FUNCTION_BLOCK "FB_FedExLoginResponse"
TITLE = FB_IDFWD
{ S7_Optimized_Access := 'TRUE' }
AUTHOR : MHSE
FAMILY : UPS_SpecificCommunication
VERSION : 3.0
// ATTRIBUTES
// AUTO_NUMBER = True
// BLOCK_NUMBER = 77
// END_ATTRIBUTES
//Function block to prepare and send the UPS IDFWD message.
   VAR_INPUT
      iUDT_Facility { ExternalAccessible := 'False'; ExternalVisible := 'False'; ExternalWritable := 'False'} : "UDT_FedExFacility";   // System configuration
      is_LastHost { ExternalAccessible := 'False'; ExternalVisible := 'False'; ExternalWritable := 'False'} : String;   // IP Address of the existing connection. If this isthe first connection, IP Address or Hostname
      ix_ConnectionStatus { ExternalAccessible := 'False'; ExternalVisible := 'False'; ExternalWritable := 'False'} : Bool;   // 1- Success, 0- Failure
   END_VAR

   VAR_OUTPUT
      qx_Error { ExternalAccessible := 'False'; ExternalVisible := 'False'; ExternalWritable := 'False'} : Bool;   // Collective error output
   END_VAR

   VAR_IN_OUT
      iqUDT_FifoHeader : "UDT_FifoHeader";   // FIFO header
      iqa_FifoData : Array[*] of "UDT_Message";   // FIFO data
   END_VAR

   VAR
      s_R_TRIG_LoginRequest {InstructionName := 'R_TRIG'; LibVersion := '1.0'; ExternalAccessible := 'False'; ExternalVisible := 'False'; ExternalWritable := 'False'; S7_SetPoint := 'False'} : R_TRIG;   // R_TRIG send login responde messge
      s_UDT_MessageArray { ExternalAccessible := 'False'; ExternalVisible := 'False'; ExternalWritable := 'False'; S7_SetPoint := 'False'} : "UDT_Message";   // Message character array
      sa_Status { ExternalAccessible := 'False'; ExternalVisible := 'False'; ExternalWritable := 'False'} : Struct   // Status structure
         FIFOStatus { ExternalAccessible := 'False'; ExternalVisible := 'False'; ExternalWritable := 'False'} : "UDT_FifoStatus";   //  FIFO Status structure
         FIFOError { ExternalAccessible := 'False'; ExternalVisible := 'False'; ExternalWritable := 'False'; S7_SetPoint := 'True'} : Bool;   //  FIFO error
         FIFOWarning { ExternalAccessible := 'False'; ExternalVisible := 'False'; ExternalWritable := 'False'; S7_SetPoint := 'True'} : Bool;   //  FIFO warning
         InvalidSystemIDLen { ExternalAccessible := 'False'; ExternalVisible := 'False'; ExternalWritable := 'False'} : Bool;   //  Invalid designated system parameter input
         InvalidFacialityIDLen { ExternalAccessible := 'False'; ExternalVisible := 'False'; ExternalWritable := 'False'} : Bool;   //  Invalid GIN
         InvalidMsgArraySize { ExternalAccessible := 'False'; ExternalVisible := 'False'; ExternalWritable := 'False'} : Bool;   //  Invalid message array size
      END_STRUCT;
      ss_Message { ExternalAccessible := 'False'; ExternalVisible := 'False'; ExternalWritable := 'False'} : String;   // Message character string
      ss_ConnectionStatus { ExternalAccessible := 'False'; ExternalVisible := 'False'; ExternalWritable := 'False'} : String;   // Connection status. Y- Sucess, N- Failure
      ss_LastHost { ExternalAccessible := 'False'; ExternalVisible := 'False'; ExternalWritable := 'False'} : String;   // Last host IP adress
      ss_VersionID { ExternalAccessible := 'False'; ExternalVisible := 'False'; ExternalWritable := 'False'} : String;   // Version ID
      sui_MsgArrayElNr { ExternalAccessible := 'False'; ExternalVisible := 'False'; ExternalWritable := 'False'} : UInt;   // Number of written message characters
      si_MaxMsgLen { ExternalAccessible := 'False'; ExternalVisible := 'False'; ExternalWritable := 'False'} : Int;   // Maximum message length
      si_MsgLen { ExternalAccessible := 'False'; ExternalVisible := 'False'; ExternalWritable := 'False'} : Int;   // String character message length
      si_FacialityIDLen { ExternalAccessible := 'False'; ExternalVisible := 'False'; ExternalWritable := 'False'} : Int;   // Faciality ID length
      si_SystemIDLen { ExternalAccessible := 'False'; ExternalVisible := 'False'; ExternalWritable := 'False'} : Int;   // System ID length
      si_VersionIDLen { ExternalAccessible := 'False'; ExternalVisible := 'False'; ExternalWritable := 'False'} : Int;   // Version ID length
      si_i { ExternalAccessible := 'False'; ExternalVisible := 'False'; ExternalWritable := 'False'} : Int;   // Loop counter
      si_LastHostLen { ExternalAccessible := 'False'; ExternalVisible := 'False'; ExternalWritable := 'False'} : Int;   // Last host field length
      si_j { ExternalAccessible := 'False'; ExternalVisible := 'False'; ExternalWritable := 'False'} : Int;   // Loop counter
   END_VAR

   VAR CONSTANT
      cc_NULL : Char := '$00';   // NULL sign
      cc_STX : Char := '$02';   // Message type
      cc_ETX : Char := '$03';   // End of the text
      cs_MessageLength : String := '0066';   // Start of the text
      cs_MessageType : String := 'LR';   // Legth of the message
   END_VAR


BEGIN
	(*
	----------------------------------------------------------------------------------------

	Version history:
	Date        | Version   | Author        | Remark
	----------------------------------------------------------------------------------------
	30/06/2021  | 1.0       | J.Krawczuk    | first release MHS TIA 16.0
	16/11/2021  | 1.2       | M.Piela       | Updating regions numbering and interface changes
	21/02/2023  | 4.0       | F.Baten       | 4.0 Release TIA 17.5
	*)

	REGION 1 – FIFO header status update

	    // Mode 'S' - FIFO register status update
	    "FC_Fifo"(ic_Mode := 'S',
	              qUDT_Status => #sa_Status.FIFOStatus,
	              qx_Error => #sa_Status.FIFOError,
	              qx_Warning => #sa_Status.FIFOWarning,
	              iqv_Data := #s_UDT_MessageArray,
	              iqUDT_FifoHeader := #iqUDT_FifoHeader,
	              iqv_DataBuffer := #iqa_FifoData);

	END_REGION

	REGION 2 – Configuration check and create error

	    #si_FacialityIDLen := LEN(#iUDT_Facility.FacilityID);
	    #si_SystemIDLen := LEN(#iUDT_Facility.SystemID);

	    #sa_Status.InvalidSystemIDLen := #si_SystemIDLen <> 15;
	    #sa_Status.InvalidFacialityIDLen := #si_FacialityIDLen <> 6;

	END_REGION

	REGION 3 – Message preparation


	    IF (NOT #iqUDT_FifoHeader.Status.Full)                         // FIFO isn't full
	    THEN
	        IF (NOT #sa_Status.FIFOError                                // No FIFO errors
	            AND NOT #sa_Status.InvalidSystemIDLen                   // Length of system ID field is ok
	            AND NOT #sa_Status.InvalidFacialityIDLen)               // Length of faciality ID field is ok

	        THEN
	            REGION 3.1 – Message preparation

	                IF #ix_ConnectionStatus                             //Creating connection status
	                THEN
	                    #ss_ConnectionStatus := 'Y';

	                ELSE
	                    #ss_ConnectionStatus := 'N';

	                END_IF;

	                #ss_LastHost := '';                                 // Initializing Last host field
	                #ss_LastHost := #is_LastHost;
	                #si_LastHostLen := LEN(#ss_LastHost);

	                // Filling up rest of the field with spaces
	                FOR #si_i := 1 TO 32 - #si_LastHostLen DO

	                    #ss_LastHost := CONCAT(IN1 := #ss_LastHost,
	                                           IN2 := ' ');

	                END_FOR;

	                #ss_VersionID := '';                                // Initializing Version ID field
	                #ss_VersionID := #iUDT_Facility.VersionID;
	                #si_VersionIDLen := LEN(#ss_VersionID);

	                // Filling up rest of the field with space
	                FOR #si_j := 1 TO 6 - #si_VersionIDLen DO

	                    #ss_VersionID := CONCAT(IN1 := #ss_VersionID,
	                                            IN2 := ' ');

	                END_FOR;

	                // Message preparation

	                // Login Response message composing according to the structure
	                #ss_Message := CONCAT(IN1 := #cc_STX,                               // Start of the message (STX) '$02'
	                                      IN2 := #cs_MessageLength,                     // Message length
	                                      IN3 := #cs_MessageType,                       // Message type
	                                      IN4 := #iUDT_Facility.FacilityID,           // Facility ID
	                                      IN5 := #iUDT_Facility.SystemID,             // System ID
	                                      IN6 := #ss_VersionID,                         // Used version ID
	                                      IN7 := #ss_ConnectionStatus,                  // Connection status
	                                      IN8 := #ss_LastHost,                          // Last connected host IP adress
	                                      IN9 := #cc_ETX);                              // End of the message (ETX) '$03"

	            END_REGION

	            REGION 3.2 – Maximum number of the message characters

	                #si_MaxMsgLen := "FC_GetNrOfArrayEl"(iv_Array := #s_UDT_MessageArray.Character);

	            END_REGION

	            REGION 3.3 – Length of the complete message

	                #si_MsgLen := LEN(#ss_Message);

	            END_REGION

	            REGION 3.4 –  Message array size validation

	                #sa_Status.InvalidMsgArraySize := #si_MsgLen > #si_MaxMsgLen;

	            END_REGION

	            REGION 3.5 –  Message character string conversion to a message array of characters

	                IF (NOT #sa_Status.InvalidMsgArraySize)                 // Message character array size is valid
	                THEN

	                    Strg_TO_Chars(Strg := #ss_Message,
	                                  pChars := 0,
	                                  Cnt => #sui_MsgArrayElNr,
	                                  Chars := #s_UDT_MessageArray.Character);

	                END_IF;

	            END_REGION

	            REGION 3.6 – Clearing remaining characters in the message character array

	                IF (NOT #sa_Status.InvalidMsgArraySize)                 // Message character array size is valid
	                THEN

	                    // Filling up not used message character array elements with ' '
	                    FILL_BLK(IN := #cc_NULL,
	                             COUNT := UINT_TO_ULINT(INT_TO_UINT(#si_MaxMsgLen) - #sui_MsgArrayElNr),
	                             OUT => #s_UDT_MessageArray.Character[#sui_MsgArrayElNr]);

	                END_IF;

	            END_REGION


	            REGION 3.7 – Message write into a FIFO register

	                IF (NOT #sa_Status.InvalidMsgArraySize)      // Message character array size is valid
	                THEN

	                    // Mode 'W' - Write FIFO record
	                    "FC_Fifo"(ic_Mode := 'W',
	                              qUDT_Status => #sa_Status.FIFOStatus,
	                              qx_Error => #sa_Status.FIFOError,
	                              qx_Warning => #sa_Status.FIFOWarning,
	                              iqv_Data := #s_UDT_MessageArray,
	                              iqUDT_FifoHeader := #iqUDT_FifoHeader,
	                              iqv_DataBuffer := #iqa_FifoData);

	                END_IF;

	            END_REGION

	        END_IF;

	        // In case of FIFO full, the FIFO full error bit and FIFO collective error bit are set
	    ELSE
	        #sa_Status.FIFOError := TRUE;
	        #sa_Status.FIFOStatus.FifoFull := TRUE;

	    END_IF;

	END_REGION

	REGION 4 – Status

	    // Parametrization collective error output
	    #qx_Error :=
	    #sa_Status.InvalidSystemIDLen                               // Invalid System ID string length
	    OR #sa_Status.InvalidFacialityIDLen                         // Invalid Faciality ID lenght
	    OR #sa_Status.InvalidMsgArraySize                           // Invalid message array size
	    OR #sa_Status.FIFOError;                                    // FIFO error

	END_REGION
END_FUNCTION_BLOCK

FUNCTION_BLOCK "FB_FedExEquipmentStatusMessage"
TITLE = FB_Heartbeat
{ S7_Optimized_Access := 'TRUE' }
AUTHOR : MHSE
FAMILY : UPS_SpecificCommunication
VERSION : 3.0
// ATTRIBUTES
// AUTO_NUMBER = True
// BLOCK_NUMBER = 72
// END_ATTRIBUTES
//Function block to send and monitor the UPS heartbeat message.
   VAR_INPUT
      iUDT_Facility { ExternalAccessible := 'False'; ExternalVisible := 'False'; ExternalWritable := 'False'} : "UDT_FedExFacility";   // System configuration
      is_LOConEquipment { ExternalAccessible := 'False'; ExternalVisible := 'False'; ExternalWritable := 'False'} : String[3];   // Location of the equipment
      is_DEPCOD { ExternalAccessible := 'False'; ExternalVisible := 'False'; ExternalWritable := 'False'} : String[6];   // Depot Code
      is_TYPofEquipment { ExternalAccessible := 'False'; ExternalVisible := 'False'; ExternalWritable := 'False'} : String[3];   // Type of equipment
      is_NumberOfTheEquipment { ExternalAccessible := 'False'; ExternalVisible := 'False'; ExternalWritable := 'False'} : String[3];   // Number of the equipment 001-999
      is_DeviceType { ExternalAccessible := 'False'; ExternalVisible := 'False'; ExternalWritable := 'False'} : String[6];   // Type of Device
      is_DeviceID { ExternalAccessible := 'False'; ExternalVisible := 'False'; ExternalWritable := 'False'} : String[6];   // ID of the Device Type
      is_StatusCode { ExternalAccessible := 'False'; ExternalVisible := 'False'; ExternalWritable := 'False'} : String[3];   // Status code values
   END_VAR

   VAR_OUTPUT
      qx_Error { ExternalAccessible := 'False'; ExternalVisible := 'False'; ExternalWritable := 'False'} : Bool;   // Error
   END_VAR

   VAR_IN_OUT
      iqUDT_FifoHeader : "UDT_FifoHeader";   // FIFO header
      iqa_FifoData : Array[*] of "UDT_Message";   // FIFO data
   END_VAR

   VAR
      sUDT_MessageArray { ExternalAccessible := 'False'; ExternalVisible := 'False'; ExternalWritable := 'False'; S7_SetPoint := 'False'} : "UDT_Message";   // Message character array
      sa_Status { ExternalAccessible := 'False'; ExternalVisible := 'False'; ExternalWritable := 'False'} : Struct   // Status structure
         FIFOStatus { ExternalAccessible := 'False'; ExternalVisible := 'False'; ExternalWritable := 'False'} : "UDT_FifoStatus";   // FIFO status structure
         FIFOError { ExternalAccessible := 'False'; ExternalVisible := 'False'; ExternalWritable := 'False'; S7_SetPoint := 'True'} : Bool;   // FIFO data buffer full
         FIFOWarning { ExternalAccessible := 'False'; ExternalVisible := 'False'; ExternalWritable := 'False'; S7_SetPoint := 'True'} : Bool;   // FIFO error
         InvalidGIN { ExternalAccessible := 'False'; ExternalVisible := 'False'; ExternalWritable := 'False'} : Bool;   //  Invalid GIN
         InvalidMessageLength { ExternalAccessible := 'False'; ExternalVisible := 'False'; ExternalWritable := 'False'} : Bool;   //  Invalid PLC ID or TRAY ID
         InvalidMsgArraySize { ExternalAccessible := 'False'; ExternalVisible := 'False'; ExternalWritable := 'False'} : Bool;   // Heartbeat timeout lower than zero or lower than heartbeat time interval
      END_STRUCT;
      ss_LLCSystemID { ExternalAccessible := 'False'; ExternalVisible := 'False'; ExternalWritable := 'False'} : String[15];   // Identifier of Low-Level controls
      ss_DeviceID { ExternalAccessible := 'False'; ExternalVisible := 'False'; ExternalWritable := 'False'} : String[6];
      ss_DeviceType { ExternalAccessible := 'False'; ExternalVisible := 'False'; ExternalWritable := 'False'} : String[6];
      ss_StatusCode { ExternalAccessible := 'False'; ExternalVisible := 'False'; ExternalWritable := 'False'} : String[3];
      ss_Message { ExternalAccessible := 'False'; ExternalVisible := 'False'; ExternalWritable := 'False'} : String;   // Message character string
      sui_MsgArrayElNr { ExternalAccessible := 'False'; ExternalVisible := 'False'; ExternalWritable := 'False'} : UInt;   // Invalid message array size
      si_MaxMsgLen { ExternalAccessible := 'False'; ExternalVisible := 'False'; ExternalWritable := 'False'} : Int;   // Maximum message length
      si_MsgLen { ExternalAccessible := 'False'; ExternalVisible := 'False'; ExternalWritable := 'False'} : Int;   // String character message length
      si_LostMsg { ExternalAccessible := 'False'; ExternalVisible := 'False'; ExternalWritable := 'False'} : Int;   // Number of lost messages
      si_DeviceIDLen { ExternalAccessible := 'False'; ExternalVisible := 'False'; ExternalWritable := 'False'} : Int;
      si_DeviceTypeLen { ExternalAccessible := 'False'; ExternalVisible := 'False'; ExternalWritable := 'False'} : Int;
      si_StatusCodeLen { ExternalAccessible := 'False'; ExternalVisible := 'False'; ExternalWritable := 'False'} : Int;
      si_LenFillLoop { ExternalAccessible := 'False'; ExternalVisible := 'False'; ExternalWritable := 'False'} : Int;   // Loop couter
      sx_MsgLost { ExternalAccessible := 'False'; ExternalVisible := 'False'; ExternalWritable := 'False'} : Bool;   // Message lost
   END_VAR

   VAR CONSTANT
      cc_NULL : Char := '$00';   // NULL sign
      cc_STX : Char := '$02';   // Start of the text
      cc_ETX : Char := '$03';   // End of the text
      cs_Length : String := '0058';   // Legth of the message
      cs_MessageType : String := 'ES';   // Message type
   END_VAR


BEGIN
	(*
	----------------------------------------------------------------------------------------

	Version history:
	Date        | Version   | Author        | Remark
	----------------------------------------------------------------------------------------
	24/05/2019  | 0.1       | L.Klar        | first release MHS TIA 15.1
	29/06/2021  | 1.0       | F.Baten       | first release MHS TIA 16.4
	10/11/2021  | 1.2       | M.Piela       | Updating regions numbering, interface changes
	10/11/2021  | 1.3       | M.Piela       | Device ID, Device Type and Status Code conversion
	21/02/2023  | 4.0       | F.Baten       | 4.0 Release TIA 17.5
	*)

	REGION 1 – FIFO header status update

	    // Mode 'S' - FIFO register status update
	    "FC_Fifo"(ic_Mode := 'S',
	              qUDT_Status => #sa_Status.FIFOStatus,
	              qx_Error => #sa_Status.FIFOError,
	              qx_Warning => #sa_Status.FIFOWarning,
	              iqv_Data := #sUDT_MessageArray,
	              iqUDT_FifoHeader := #iqUDT_FifoHeader,
	              iqv_DataBuffer := #iqa_FifoData);
	END_REGION

	REGION 2 – Message preparation

	    IF NOT #iqUDT_FifoHeader.Status.Full                 // FIFO isn't full
	    THEN

	        REGION 2.1 - LLC System ID
	            #ss_LLCSystemID := CONCAT(IN1 := #is_DEPCOD,
	                                      IN2 := #is_LOConEquipment,
	                                      IN3 := #is_TYPofEquipment,
	                                      IN4 := #is_NumberOfTheEquipment);
	        END_REGION

	        REGION 2.2. Device Type

	            #ss_DeviceType := #is_DeviceType;
	            #si_DeviceTypeLen := LEN(#ss_DeviceType);

	            IF #si_DeviceTypeLen < 6
	            THEN
	                FOR #si_LenFillLoop := #si_DeviceTypeLen TO 6 DO
	                    #ss_DeviceType := CONCAT(IN1 := #ss_DeviceType,
	                                             IN2 := ' ');
	                END_FOR;

	            END_IF;

	        END_REGION

	        REGION 2.3. Device ID

	            #ss_DeviceID := #is_DeviceID;
	            #si_DeviceIDLen := LEN(#ss_DeviceID);

	            IF #si_DeviceIDLen < 6
	            THEN
	                FOR #si_LenFillLoop := #si_DeviceIDLen TO 6 DO
	                    #ss_DeviceID := CONCAT(IN1 := #ss_DeviceID,
	                                           IN2 := ' ');
	                END_FOR;

	            END_IF;

	        END_REGION

	        REGION 2.4. Status Code

	            #ss_StatusCode := #is_StatusCode;
	            #si_StatusCodeLen := LEN(#ss_StatusCode);

	            IF #si_StatusCodeLen < 3
	            THEN
	                FOR #si_LenFillLoop := #si_StatusCodeLen TO 3 DO
	                    #ss_StatusCode := CONCAT(IN1 := #ss_StatusCode,
	                                             IN2 := ' ');
	                END_FOR;

	            END_IF;

	        END_REGION

	        IF NOT #sa_Status.FIFOError                   // No FIFO error
	        THEN
	            REGION 2.5 – Message preparation
	                // Message composing according to the structure: STX,Body ,ETX
	                #ss_Message := CONCAT(IN1 := #cc_STX,
	                                      IN2 := #cs_Length,
	                                      IN3 := #cs_MessageType,
	                                      IN4 := #ss_LLCSystemID,
	                                      IN5 := #ss_DeviceType,
	                                      IN6 := #ss_DeviceID,
	                                      IN7 := #ss_StatusCode,
	                                      IN8 := "DB_Time".Timestamp,
	                                      IN9 := #iUDT_Facility.TimeZoneDesignator,
	                                      IN10 := #cc_ETX);

	            END_REGION

	            REGION 2.6 – Maximum number of the message characters

	                #si_MaxMsgLen := "FC_GetNrOfArrayEl"(iv_Array := #sUDT_MessageArray.Character);

	            END_REGION

	            REGION 2.7 – Length of the complete message

	                #si_MsgLen := LEN(#ss_Message);
	                // Message length validation
	                #sa_Status.InvalidMessageLength := #si_MsgLen - 2 <> STRING_TO_INT(#cs_Length);

	            END_REGION

	            REGION 2.8 –  Message array size validation

	                #sa_Status.InvalidMsgArraySize := #si_MsgLen > #si_MaxMsgLen;

	            END_REGION

	            REGION 2.9 –  Message character string conversion to a message array of characters

	                IF (NOT #sa_Status.InvalidMsgArraySize)     // Message character array size is valid
	                THEN

	                    Strg_TO_Chars(Strg := #ss_Message,
	                                  pChars := 0,
	                                  Cnt => #sui_MsgArrayElNr,
	                                  Chars := #sUDT_MessageArray.Character);

	                END_IF;

	            END_REGION

	            REGION 2.10 – Clearing remaining characters in the message character array

	                IF (NOT #sa_Status.InvalidMsgArraySize)     // Message character array size is valid
	                THEN

	                    // Filling up not used message character array elements with '$00' (ASCII - 16#00)
	                    FILL_BLK(IN := #cc_NULL,
	                             COUNT := UINT_TO_ULINT(INT_TO_UINT(#si_MaxMsgLen) - #sui_MsgArrayElNr),
	                             OUT => #sUDT_MessageArray.Character[#sui_MsgArrayElNr]);

	                END_IF;

	            END_REGION

	            REGION 2.11 – Message write into a FIFO register

	                IF NOT #sa_Status.InvalidMsgArraySize      // Message character array size is valid
	                THEN

	                    // Mode 'W' - Write FIFO record
	                    "FC_Fifo"(ic_Mode := 'W',
	                              qUDT_Status => #sa_Status.FIFOStatus,
	                              qx_Error => #sa_Status.FIFOError,
	                              qx_Warning => #sa_Status.FIFOWarning,
	                              iqv_Data := #sUDT_MessageArray,
	                              iqUDT_FifoHeader := #iqUDT_FifoHeader,
	                              iqv_DataBuffer := #iqa_FifoData);
	                END_IF;

	            END_REGION

	        END_IF;

	        // In case of FIFO full, the FIFO full error bit and FIFO collective error bit are set
	    ELSE

	        #sa_Status.FIFOError := TRUE;
	        #sa_Status.FIFOStatus.FifoFull := TRUE;

	    END_IF;

	END_REGION

	REGION 3 - Writing output

	    #qx_Error := #sa_Status.InvalidMessageLength        // Invalid message length
	    OR #sa_Status.InvalidMsgArraySize                   // Invalid message array size
	    OR #sa_Status.FIFOError;                            // FIFO error

	END_REGION
END_FUNCTION_BLOCK

FUNCTION "FC_Statistics" : Void
TITLE = FC_Statistics
{ S7_Optimized_Access := 'TRUE' }
AUTHOR : MHSE
FAMILY : GeneralSystemFunctions
VERSION : 3.0
// ATTRIBUTES
// AUTO_NUMBER = True
// BLOCK_NUMBER = 26
// END_ATTRIBUTES
//Function to calculate statistics.
   VAR_INPUT
      ix_Reset : Bool;   // Reset statistics data
      ix_Activate : Bool;   // Activete statistics counters
      ix_RTrigActivate : Bool;   // Activation rise trigger
   END_VAR

   VAR_IN_OUT
      iqUDT_Statistics : "UDT_EventStatistic";   // Statistic structure
   END_VAR


BEGIN
	(*
	----------------------------------------------------------------------------------------

	Version history:
	Date        | Version   | Author        | Remark
	----------------------------------------------------------------------------------------
	24/05/2019  | 0.1       | C. Leite      | first release MHS TIA 15.1
	17/07/2019  | 0.2       | A.Nowak       | Add comments
	24/07/2019  | 2.0       | L.Klar        | 2.0 MHS library release TIA 15.1
	27/08/2019  | 2.1       | M.Kurpiers    | Comments adjusted
	04/11/2019  | 2.2       | L.Klar        | 1 second pulse changed from memory bit to DB variable
	12/11/2019  | 3.0       | P.Majka       | 3.0 MHS library release TIA 15.1
	21/02/2023  | 4.0       | F.Baten       | 4.0 Release TIA 17.5
	*)

	REGION 1 - Number of events

	    IF (#ix_RTrigActivate)      // Event occured
	    THEN

	        // Increment the number of times the event occurred and clear the time of the current or last event
	        #iqUDT_Statistics.NumberOfTimes += 1;
	        #iqUDT_Statistics.LastEventSeconds := 0;

	    END_IF;

	END_REGION

	REGION 2 - Event time

	    // 1 shot every 1 sec and activate statistic counter
	    IF ("DB_Memory".OS_1sec AND #ix_Activate)
	    THEN

	        // Increment the time of the current or last event and the time of all events that occured
	        #iqUDT_Statistics.LastEventSeconds += 1;
	        #iqUDT_Statistics.TotalEventSeconds += 1;

	    END_IF;

	END_REGION

	REGION 3 - Data reset


	    IF (#ix_Reset)                                            // Reset statistics data
	    THEN

	        IF (NOT #ix_Activate)                                 // Statistic counter isn't activate
	        THEN

	            // Clear statistics data
	            #iqUDT_Statistics.NumberOfTimes := 0;
	            #iqUDT_Statistics.LastEventSeconds := 0;
	            #iqUDT_Statistics.TotalEventSeconds := 0;

	        ELSE

	            // Write 1 to the number of times the event occurred and clear times
	            #iqUDT_Statistics.NumberOfTimes := 1;
	            #iqUDT_Statistics.LastEventSeconds := 0;
	            #iqUDT_Statistics.TotalEventSeconds := 0;

	        END_IF;

	    END_IF;

	END_REGION
END_FUNCTION

FUNCTION_BLOCK "FB_PneumaticBrakeUnit"
TITLE = FB_PneumaticBrakeUnit
{ S7_Optimized_Access := 'TRUE' }
AUTHOR : 'F.Baten'
VERSION : 0.1
// ATTRIBUTES
// AUTO_NUMBER = True
// BLOCK_NUMBER = 223
// END_ATTRIBUTES
//Function to control a pneumatic brake contol
   VAR_INPUT
      iUDT_PneumaticBreakConfiguration { ExternalAccessible := 'False'; ExternalVisible := 'False'; ExternalWritable := 'False'} : "UDT_PneumaticBrakeConfiguration";   // Pneumatic brake configuration structure
      ix_PECBrake { ExternalAccessible := 'False'; ExternalVisible := 'False'; ExternalWritable := 'False'} : Bool;   // TRUE when the brake photoye is not blocked
      ix_PECStop { ExternalAccessible := 'False'; ExternalVisible := 'False'; ExternalWritable := 'False'} : Bool;   // TRUE when the stop photoye is not blocked
      ix_PECdownstream { ExternalAccessible := 'False'; ExternalVisible := 'False'; ExternalWritable := 'False'} : Bool;   // TRUE when the photoye downstream is not blocked
      ix_DownstreamStopActive { ExternalAccessible := 'False'; ExternalVisible := 'False'; ExternalWritable := 'False'} : Bool;   // TRUE when the downstream stop is active
      ix_MasterValve { ExternalAccessible := 'False'; ExternalVisible := 'False'; ExternalWritable := 'False'} : Bool;   // TRUE when master valve is on
      ix_SafetyOk { ExternalAccessible := 'False'; ExternalVisible := 'False'; ExternalWritable := 'False'} : Bool;   // TRUE when safety is ok
   END_VAR

   VAR_OUTPUT
      qx_Valve { ExternalAccessible := 'False'; ExternalVisible := 'False'; ExternalWritable := 'False'} : Bool;   // TRUE when valve is activated
      qx_StopActive { ExternalAccessible := 'False'; ExternalVisible := 'False'; ExternalWritable := 'False'} : Bool;   // TRUE when stop is activated to upstream
   END_VAR

   VAR_IN_OUT
      iqUDT_EquipmentControl : "UDT_EquipmentControl";   // Equipment control structure
   END_VAR

   VAR
      s_PECBreakTimerOnOffDelay { ExternalAccessible := 'False'; ExternalVisible := 'False'; ExternalWritable := 'False'; S7_SetPoint := 'False'} : "FB_TimerOnOffDelay";   // Filtering end of section photo eye signal
      s_PECStopTimerOnOffDelay { ExternalAccessible := 'False'; ExternalVisible := 'False'; ExternalWritable := 'False'; S7_SetPoint := 'False'} : "FB_TimerOnOffDelay";   // Filtering end of section photo eye signal
      s_StopFunctionTimerOnOffDelay { ExternalAccessible := 'False'; ExternalVisible := 'False'; ExternalWritable := 'False'; S7_SetPoint := 'False'} : "FB_TimerOnOffDelay";   // Filtering end of section photo eye signal
      s_StopReleaseOnOffDelay { ExternalAccessible := 'False'; ExternalVisible := 'False'; ExternalWritable := 'False'; S7_SetPoint := 'False'} : "FB_TimerOnOffDelay";
      sR_TRIG_PECStop {InstructionName := 'R_TRIG'; LibVersion := '1.0'; ExternalAccessible := 'False'; ExternalVisible := 'False'; ExternalWritable := 'False'; S7_SetPoint := 'False'} : R_TRIG;   // Rising edge trigger PEC jam
      slr_StepTimer { ExternalAccessible := 'False'; ExternalVisible := 'False'; ExternalWritable := 'False'} : LReal;   // Step timer
      slr_BrakeInterval { ExternalAccessible := 'False'; ExternalVisible := 'False'; ExternalWritable := 'False'} : LReal;   // Brake interval
      si_BrakeFunction { ExternalAccessible := 'False'; ExternalVisible := 'False'; ExternalWritable := 'False'} : Int;   // Brake function step
      si_BrakeCycles { ExternalAccessible := 'False'; ExternalVisible := 'False'; ExternalWritable := 'False'} : Int;   // Number of cyles
      sx_Cycle { ExternalAccessible := 'False'; ExternalVisible := 'False'; ExternalWritable := 'False'} : Bool;   // Cycle
      sx_PECBrakeFiltered { ExternalAccessible := 'False'; ExternalVisible := 'False'; ExternalWritable := 'False'} : Bool;   // PEC signal filtered
      sx_PECStopFiltered { ExternalAccessible := 'False'; ExternalVisible := 'False'; ExternalWritable := 'False'} : Bool;   // PEC signal filtered
      sx_DownstreamStop { ExternalAccessible := 'False'; ExternalVisible := 'False'; ExternalWritable := 'False'} : Bool;   // Downstream is stopped
      sx_StopFunctionActive { ExternalAccessible := 'False'; ExternalVisible := 'False'; ExternalWritable := 'False'} : Bool;   // Stop function is activated
      sx_BrakePulse { ExternalAccessible := 'False'; ExternalVisible := 'False'; ExternalWritable := 'False'} : Bool;   // Brake pulse 1 is active
      sx_BrakeAssemblyValve { ExternalAccessible := 'False'; ExternalVisible := 'False'; ExternalWritable := 'False'} : Bool;   // Brake assembly valve
      sx_NoCycles { ExternalAccessible := 'False'; ExternalVisible := 'False'; ExternalWritable := 'False'} : Bool;   // No cycles
      sx_Enable_release { ExternalAccessible := 'False'; ExternalVisible := 'False'; ExternalWritable := 'False'} : Bool;
   END_VAR

   VAR CONSTANT
      ci_ReleaseStopBreakTimeOnDelay : UInt := 10000;
   END_VAR


BEGIN
	(*
	----------------------------------------------------------------------------------------

	Version history:
	Date        | Version   | Author        | Remark
	----------------------------------------------------------------------------------------
	23/06/2021  | 0.0       | F. Baten      | first release TIA 15.1
	20/10/2021  | 0.1       | M. Piela      | Add equipment control. Stylistic correction
	25/06/2021  | 0.2       | M. Kurpiers   | Add stop break release
	21/02/2023  | 4.0       | F.Baten       | 4.0 Release TIA 17.5
	 *)

	REGION 1 - Timers

	    // Filtering brake photo eye signal
	    #s_PECBreakTimerOnOffDelay(iudi_OnDelayTime := #iUDT_PneumaticBreakConfiguration.PECBrakeOnDelay,
	                               iudi_OffDelayTime := #iUDT_PneumaticBreakConfiguration.PECBrakeOffDelay,
	                               ix_SignalToDelay := #ix_PECBrake,
	                               ix_Enable := TRUE,
	                               qx_DelayedSignal => #sx_PECBrakeFiltered);

	    // Filtering stop photo eye signal
	    #s_PECStopTimerOnOffDelay(iudi_OnDelayTime := #iUDT_PneumaticBreakConfiguration.PECStopOnDelay,
	                              iudi_OffDelayTime := #iUDT_PneumaticBreakConfiguration.PECStopOffDelay,
	                              ix_SignalToDelay := #ix_PECStop,
	                              ix_Enable := TRUE,
	                              qx_DelayedSignal => #sx_PECStopFiltered);

	    // Filtering downstream stop photo eye signal
	    #s_StopFunctionTimerOnOffDelay(iudi_OnDelayTime := #iUDT_PneumaticBreakConfiguration.StopFunctionOnDelay,
	                                   iudi_OffDelayTime := #iUDT_PneumaticBreakConfiguration.StopFunctionOffDelay,
	                                   ix_SignalToDelay := #ix_DownstreamStopActive,
	                                   ix_Enable := TRUE,
	                                   qx_DelayedSignal => #sx_DownstreamStop);

	    #s_StopReleaseOnOffDelay(iudi_OnDelayTime := #ci_ReleaseStopBreakTimeOnDelay,
	                             iudi_OffDelayTime := 0,
	                             ix_SignalToDelay := #ix_PECdownstream AND NOT #ix_PECBrake,
	                             ix_Enable := TRUE,
	                             qx_DelayedSignal => #sx_Enable_release);

	    // Sequence Timer
	    IF #slr_StepTimer > 0
	    THEN
	        #slr_StepTimer -= "DB_Memory".PrevCycleTime;
	        IF #slr_StepTimer < 0
	        THEN
	            #slr_StepTimer := 0;
	        END_IF;
	    END_IF;

	END_REGION

	REGION 2 - Brake function
	    // Braking of the parcel is activated when first parcel arrives in brake PEC and stop function is not active.
	    // Now the brake is raised configured number of times with the configured brakepuls time and the configured delay. this is done every time again with the configured
	    // interval time as long as the PEC brake is occupied.

	    #sR_TRIG_PECStop(CLK := #ix_PECStop);
	    // Restart sequence
	    IF #sR_TRIG_PECStop.Q AND NOT #sx_PECStopFiltered
	    THEN
	        #si_BrakeFunction := 1;
	    END_IF;

	    IF #sx_NoCycles AND #ix_PECBrake THEN
	        #sx_NoCycles := FALSE;
	    END_IF;

	    IF #iUDT_PneumaticBreakConfiguration.BrakeCycles = 1
	    THEN
	        #slr_BrakeInterval := #iUDT_PneumaticBreakConfiguration.BrakePause;
	    ELSE
	        #slr_BrakeInterval := #iUDT_PneumaticBreakConfiguration.BrakeInterval;
	    END_IF;
	    // Sequence
	    IF #si_BrakeFunction = 1 AND #slr_StepTimer = 0 AND (NOT #ix_PECBrake OR #sx_BrakePulse)
	    THEN
	        #sx_BrakePulse := TRUE;
	        #slr_StepTimer := #iUDT_PneumaticBreakConfiguration.BrakePuls;
	        #si_BrakeFunction := 2;
	        #sx_Cycle := TRUE;
	    END_IF;

	    IF (#si_BrakeFunction = 2 OR #sx_Enable_release) AND #slr_StepTimer = 0 AND #ix_SafetyOk
	    THEN
	        #sx_BrakePulse := False;
	        #si_BrakeCycles += 1;
	        IF #iUDT_PneumaticBreakConfiguration.BrakeCycles > 0
	        THEN
	            IF #si_BrakeCycles >= #iUDT_PneumaticBreakConfiguration.BrakeCycles
	            THEN
	                #si_BrakeCycles := 0;
	                #slr_StepTimer := #slr_BrakeInterval;
	                #si_BrakeFunction := 3;
	                #sx_Cycle := TRUE;
	            ELSE
	                #slr_StepTimer := #iUDT_PneumaticBreakConfiguration.BrakePause;
	                #si_BrakeFunction := 1;
	                #sx_Cycle := TRUE;
	            END_IF;
	        ELSE
	            #sx_NoCycles := TRUE;
	            #si_BrakeCycles := 0;
	            #si_BrakeFunction := 4;
	        END_IF;
	    END_IF;
	    // Waiting time between interval
	    IF (#si_BrakeFunction = 3 AND #slr_StepTimer = 0) OR #sx_StopFunctionActive
	    THEN
	        #si_BrakeFunction := 1;
	    END_IF;
	    // Wait for pec to clear, one puls only
	    IF (#si_BrakeFunction = 4 AND NOT #sx_NoCycles) OR #sx_StopFunctionActive
	    THEN
	        #si_BrakeFunction := 1;
	    END_IF;

	END_REGION

	REGION 3 - Brake valve

	    REGION 3.1 - Brake assembly valve function

	        IF #sx_StopFunctionActive AND NOT #sx_DownstreamStop
	        THEN
	            #sx_StopFunctionActive := FALSE;
	        END_IF;

	        IF #sx_DownstreamStop AND NOT #sx_PECStopFiltered AND NOT #sx_PECBrakeFiltered
	        THEN
	            #sx_StopFunctionActive := TRUE;
	        END_IF;

	        #sx_BrakeAssemblyValve := (#sx_StopFunctionActive
	        AND ((#iUDT_PneumaticBreakConfiguration.Slave AND #ix_MasterValve)
	        OR NOT #iUDT_PneumaticBreakConfiguration.Slave))
	        OR (NOT #sx_StopFunctionActive
	        AND #sx_BrakePulse);

	    END_REGION

	    REGION 3.2 Valve activation

	        IF #iUDT_PneumaticBreakConfiguration.FailSafe
	        THEN
	            #qx_Valve := NOT (#sx_BrakeAssemblyValve OR NOT #ix_SafetyOk);
	        ELSE
	            #qx_Valve := #sx_BrakeAssemblyValve AND #ix_SafetyOk;
	        END_IF;

	    END_REGION

	END_REGION

	REGION 4 - Stop Active

	    #qx_StopActive := #sx_StopFunctionActive AND NOT #sx_PECStopFiltered AND NOT #sx_PECBrakeFiltered;

	END_REGION
END_FUNCTION_BLOCK

TYPE "UDT_VfdKebaSystemPO"
VERSION : 0.1
   STRUCT
      ToMCAliveCount : Int;   // Motion controller is communicating
      ToMCActiveOpMode : Int;   // Operational mode request: 0 = No Operation; 1 = Auto; 2 = Manual
      ToMCControl1 : Struct   // System control 1
         Start : Bool;   // System control - Start system in auto mode
         LocalSafetyReset : Bool;   // System control - Local safety reset
         Abort : Bool;   // System control - Abort command to interrupt every movement programmed
         Spare_3 : Bool;   // System control - Spare
         Spare_4 : Bool;   // System control - Spare
         Bypass : Bool;   // System control - bypass mode
         Spare_6 : Bool;   // System control - Spare
         StressTest : Bool;   // System control - Start system in stress test mode
         Reset : Bool;   // System control - Alarm reset
         ServoON : Bool;   // System control - Power-On enable
         HomingReq : Bool;   // System control - After the poer-on in homing mode the system perform an homing
         Spare_11 : Bool;   // System control - Spare
         Spare_12 : Bool;   // System control - Spare
         Spare_13 : Bool;   // System control - Spare
         Spare_14 : Bool;   // System control - Spare
         Spare_15 : Bool;   // System control - Spare
      END_STRUCT;
      ToMCControl2 : Struct   // System control 2
         Spare_0 : Bool;   // System control - Spare
         Spare_1 : Bool;   // System control - Spare
         Ax_BeltRunFwd : Bool;   // System control - Spare
         Ax_BeltRunBkwd : Bool;   // System control - Spare
         Spare_4 : Bool;   // System control - Spare
         Spare_5 : Bool;   // System control - Spare
         Spare_6 : Bool;   // System control - Spare
         Spare_7 : Bool;   // System control - Spare
         Spare_8 : Bool;   // System control - Spare
         Spare_9 : Bool;   // System control - Spare
         Spare_10 : Bool;   // System control - Spare
         Spare_11 : Bool;   // System control - Spare
         Spare_12 : Bool;   // System control - Spare
         Spare_13 : Bool;   // System control - Spare
         Ax1_PosRight : Bool;   // System control - Motor 1 Section 1 - command for positioningon the right
         Ax1_PosLeft : Bool;   // System control - Motor 1 Section 1 - command for positioningon the left
      END_STRUCT;
      "ToMCAx[1]" : Struct   // Axis 1 control word
         Jog_Fwd : Bool;   // Axis selected control - jog forward
         Jog_Bkwd : Bool;   // Axis selected control - jog backward
         Abort : Bool;   // Axis selected control - abort eachmovement programmed
         Spare_3 : Bool;   // Axis selected control - Spare
         Spare_4 : Bool;   // Axis selected control - Fault
         Spare_5 : Bool;   // Axis selected control - Spare
         Spare_6 : Bool;   // Axis selected control - Spare
         ZeroDirectReq : Bool;   // Axis selected control - request to perform a recording of actual position with value 0 (use only and exlusively with the conveyor in midlle position)
         Reset : Bool;   // Axis selected control - reset
         Servo_ON : Bool;   // Axis selected control - power and servo On (only for axis selected, the other axes are disabled with Servo-Off)
         Homing : Bool;   // Axis selected control - request to perform an homing procedure
         PosAbs : Bool;   // Axis selected control -  request to perform an absolute positioning
         Spare_12 : Bool;   // Axis selected control - Spare
         Stop : Bool;   // Axis selected control - stop
         QuickStop : Bool;   // Axis selected control - stop for emergency
         spare_15 : Bool;   // Axis selected control - Spare
      END_STRUCT;
      "ToMCAx[1]SpeedSetpoint" : Int;   // Speed setpoint [degree/s*10]
      "ToMCAx[1]Spare2" : Int;   // Axis 1 control - Spare
      "ToMCAx[1]Spare3" : Int;   // Axis 1 control - Spare
      "ToMCAx[1]PositionSetpointRight" : Int;   // Axis 1 control - Position setpoint right [degree*10]
      "ToMCAx[1]PositionSetpointLeft" : Int;   // Axis 1 control - Position setpoint left [degree*10]
      "ToMCAx[2]" : Struct   // Axis 2 control word
         Jog_Fwd : Bool;   // Axis selected control - jog forward
         Jog_Bkwd : Bool;   // Axis selected control - jog backward
         Abort : Bool;   // Axis selected control - abort eachmovement programmed
         Spare_3 : Bool;   // Axis selected control - Spare
         Spare_4 : Bool;   // Axis selected control - Fault
         Spare_5 : Bool;   // Axis selected control - Spare
         Spare_6 : Bool;   // Axis selected control - Spare
         ZeroDirectReq : Bool;   // Axis selected control - request to perform a recording of actual position with value 0 (use only and exlusively with the conveyor in midlle position)
         Reset : Bool;   // Axis selected control - reset
         Servo_ON : Bool;   // Axis selected control - power and servo On (only for axis selected, the other axes are disabled with Servo-Off)
         Homing : Bool;   // Axis selected control - request to perform an homing procedure
         PosAbs : Bool;   // Axis selected control -  request to perform an absolute positioning
         Spare_12 : Bool;   // Axis selected control - Spare
         Stop : Bool;   // Axis selected control - stop
         QuickStop : Bool;   // Axis selected control - stop for emergency
         Direction : Bool;   // Axis selected control - Rotation direction
      END_STRUCT;
      "ToMCAx[2]SpeedSetpoint" : Int;   // Axis 2 Speed setpoint [mm/s*10]
      "ToMCAx[2]Acceleration" : Int;   // Axis 2 Acceleration [mm/s2]
      "ToMCAx[2]Deceleration" : Int;   // Axis 2 Deceleration [mm/s2]
      "ToMCAx[2]Adjustment" : Int;   // Axis 2 Speed control adjustment
      "ToMCAx[2]PositionSetpoint" : Int;   // Axis 2 control - Position setpoint for absolute or relative positioning
   END_STRUCT;

END_TYPE

FUNCTION "FC_EquipmentReport" : Void
TITLE = FC_Equipment_Report
{ S7_Optimized_Access := 'TRUE' }
AUTHOR : MHSE
FAMILY : GeneralSystemFunctions
VERSION : 3.0
// ATTRIBUTES
// AUTO_NUMBER = True
// BLOCK_NUMBER = 16
// END_ATTRIBUTES
//Function to generate equipment report.
   VAR_INPUT
      iUDT_Status : "UDT_CommonStatus";   // Status structure
   END_VAR

   VAR_IN_OUT
      iqUDT_Control : "UDT_EquipmentControl";   // Equipment control
   END_VAR


BEGIN
	(*
	----------------------------------------------------------------------------------------

	Version history:
	Date        | Version   | Author        | Remark
	----------------------------------------------------------------------------------------
	24/05/2019  | 0.1       | F.Baten       | first release MHS TIA 15.1
	17/06/2019  | 0.3       | L.Klar        | Manual mode added to "UDT_EquipmentControl"
	17/07/2019  | 0.4       | A.Nowak       | Add all statuses and comments
	24/07/2019  | 2.0       | L.Klar        | 2.0 MHS library release TIA 15.1
	27/08/2019  | 2.1       | K.Pokorski    | Comments adjusted
	16/09/2019  | 2.2       | K.Pokorski    | Equipment error free condition added to "Restart required" status
	06/10/2019  | 2.3       | S. Deukar     | Updated accoring to new UDT equipment report
	12/11/2019  | 3.0       | P.Majka       | 3.0 MHS library release TIA 15.1
	05/02/2024  | 3.1       | L.Klar        | Auto On extention added
	13/03/2024  | 4.0       | S. Nieswiec   | Added to baseline
	*)

	REGION 1 - Equipment report update

	    // Extension of stopped equipment report with the stopped status
	    #iqUDT_Control.Report.Stopped := #iUDT_Status.Stopped
	    OR #iqUDT_Control.Report.Stopped;

	    // Extension of started equipment report with the started status
	    #iqUDT_Control.Report.Running := #iUDT_Status.Running
	    OR #iqUDT_Control.Report.Running;

	    // Extension of energy save equipment report with the energy save status
	    #iqUDT_Control.Report.EnergySave := #iUDT_Status.EnergySave
	    OR #iqUDT_Control.Report.EnergySave;

	    // Extension of warning equipment report with the warning status
	    #iqUDT_Control.Report.Warning := #iUDT_Status.Warning
	    OR #iqUDT_Control.Report.Warning;

	    // Extension of manual mode equipment report with the manual mode status
	    #iqUDT_Control.Report.Manual := #iUDT_Status.Manual
	    OR #iqUDT_Control.Report.Manual;

	    // Extension of error equipment report with the error status
	    #iqUDT_Control.Report.Error := #iUDT_Status.Error
	    OR #iqUDT_Control.Report.Error;

	    // Extension of safety stop equipment report with the safety stop status
	    #iqUDT_Control.Report.SafetyStop := #iUDT_Status.SafetyStop
	    OR #iqUDT_Control.Report.SafetyStop;

	    // Extension of Auto On equipment report with the Auto On status
	    #iqUDT_Control.Report.AutoON := #iUDT_Status.AutoON
	    OR #iqUDT_Control.Report.AutoON;

	    // Extension of restart required equipment report with the restart required and no equipment error statuses
	    #iqUDT_Control.Request.RestartRequired := #iUDT_Status.Stopped
	    AND NOT #iUDT_Status.Error
	    OR #iqUDT_Control.Request.RestartRequired;

	END_REGION
END_FUNCTION

DATA_BLOCK "DB_HMIStatusConfiguration"
TITLE = DB_HMIStatusConfiguration
{ S7_Optimized_Access := 'TRUE' }
AUTHOR : MHSE
VERSION : 3.0
NON_RETAIN
   VAR
      FireAlarm : Int;   // Fire alarm active
      SafetyStop : Int;   // Safety stop error status
      Error : Int;   // Error status
      Warning : Int;   // Warning status
      ManualRun : Int;   // Manual run status
      Manual : Int;   // Manual status
      Halted : Int;   // Halted status
      Dieback : Int;   // Die back status
      Stopped : Int;   // Stopped status
      Running : Int;   // Running status
      EnergySave : Int;   // Energy save status
      CommunicationError : Int;   // Communication error status
      CBError : Int;   // CB error status
      ProfinetError : Int;   // Profinet error status
      HardwareError : Int;   // Hardware error status
      VFDNotHealthy : Int;   // VFD noth healthy status
      VFDError : Int;   // VFD error status
      PECJam : Int;   // PEC jam status
      ChuteFull : Int;   // Chute full status
      EncoderError : Int;   // Encoder error status
      TrackingError : Int;   // Tracking error status
      DimensionError : Int;   // Dimension error status
      OperationalError : Int;   // Operational error status
      AutoON : Int;   // Automatic is on
      ChuteHalfFull : Int;   // Disable by operator
      DisableByManagement : Int;   // Disable by management
      GateOpen : Int;   // Manual operated gate is open
      GateClosed : Int;   // Manual operated gate is closed
      GateClosedAndNoOperatorPresent : Int;   // Manual operated gate is closed and no operator is present
      PositionChangeOngoing : Int;   // Lifting device or arm diverter changing position
      BufferMode : Int;   // BufferMode Active
      ContinuousMode : Int;   // ContinuousMode Active
      LabbelingMode : Int;   // LabbelingMode Active
   END_VAR


BEGIN
   FireAlarm := 1;
   SafetyStop := 3;
   Error := 5;
   Warning := 7;
   ManualRun := 9;
   Manual := 11;
   Halted := 13;
   Dieback := 15;
   Stopped := 17;
   Running := 19;
   EnergySave := 21;
   CommunicationError := 23;
   CBError := 25;
   ProfinetError := 27;
   HardwareError := 29;
   VFDNotHealthy := 31;
   VFDError := 33;
   PECJam := 35;
   ChuteFull := 37;
   EncoderError := 39;
   TrackingError := 41;
   DimensionError := 43;
   OperationalError := 45;
   AutoON := 47;
   ChuteHalfFull := 49;
   DisableByManagement := 51;
   GateOpen := 53;
   GateClosed := 55;
   GateClosedAndNoOperatorPresent := 57;
   PositionChangeOngoing := 59;
   BufferMode := 61;
   ContinuousMode := 63;
   LabbelingMode := 65;

END_DATA_BLOCK

TYPE "UDT_VfdKebaSystemStatus"
VERSION : 0.1
   STRUCT
      AX1ErrorCode : Int;   // Axis 1 error code (Rotation)
      AX2ErrorCode : Int;   // Axis 2 error code (Belt)
      PNSlaveNotOnline : Bool := FALSE;   // Profinet slave is not on line
      PNSlaveError : Bool := FALSE;   // Profinet slave has an error
      Axis1InternalError : Bool := FALSE;   // Axis 1 internal error is active, see error code
      Axis2InternalError : Bool := FALSE;   // Axis 2 internal error is active, see error code
      CommunicationError : Bool := FALSE;   // Communication error
      PositioningTimeWarning : Bool := FALSE;   // Exceeded time to reach position
      PNSlaveWarning : Bool := FALSE;   // Profinet slave has a warning
      MaintenanceWarning : Bool := FALSE;   // Maintenance mode active (local control enabled)
      HomingActiveWarning : Bool := FALSE;   // Homing mode activated
      StressTestActiveWarning : Bool := FALSE;   // Stress test mode activated
      MaintenanceManualActiveWarning : Bool := FALSE;   // Manual mode in maintenance activated
   END_STRUCT;

END_TYPE

TYPE "UDT_VfdKebaSystemPI"
VERSION : 0.1
   STRUCT
      FromMCAliveCount : Int;   // Motion controller is communicating
      FromMCActiveOpMode : Int;   // Operational mode active: 0 = No Operation; 1 = Auto; 2 = Manual; 10 = Maintenance; 12 = Maintenance manual; 13 = Homing; 14 = stress test activated
      FromMCStatus1 : Struct   // System status 1
         Running : Bool;   // System status - Running
         LocalSafetyResetRequired : Bool;   // System status - Local safety reset required
         Aborted : Bool;   // System status - Current procedure or command aborted
         STO_OK : Bool;   // System status - STO on drive module 1 and 2 activated
         ECAT_error : Bool;   // System status - Ethercat fault
         PN_error : Bool;   // System status - Profinet fault
         Bypass : Bool;   // System status - Bypass mode active
         StressTestOn : Bool;   // System status - Stress test active
         ControlUnitReady : Bool;   // System status - Control unit ready for operation
         Servo_active : Bool;   // System status - Motors powered and servo active
         Homing : Bool;   // System status - Homing procedure in progress
         Homed : Bool;   // System status - Homing performed
         Fault : Bool;   // System status - Fault active
         Spare_13 : Bool;   // System status - Spare
         Ready : Bool;   // System status - Ready for operation
         Spare_15 : Bool;   // System status - Spare
      END_STRUCT;
      FromMCStatus2 : Struct   // System status 2
         SafetySwitch_1_Engaged : Bool;   // System status - Infeeding photoeye engaged signal
         SafetySwitch_2_Engaged : Bool;   // System status - Safety switch 1 engaged signal
         SafetySwitch_3_Engaged : Bool;   // System status - Safety switch 2 engaged signal
         Outfeeding_Photoeye_Engaged : Bool;   // System status - Outfeeding photoeye engaged signal
         Infeeding_Photoeye_Engaged : Bool;   // System status - Spare
         LimitSwitch_RH_Engaged : Bool;   // System status - Limit switch RH egaged signal
         LimitSwitch_LH_Engaged : Bool;   // System status - Limit switch LH egaged signal
         HomeSwitch_Engaged : Bool;   // System status - Home switch egaged signal
         Spare_8 : Bool;   // System status - Spare
         Spare_9 : Bool;   // System status - Spare
         Spare_10 : Bool;   // System status - Spare
         Spare_11 : Bool;   // System status - Spare
         Spare_12 : Bool;   // System status - Spare
         Spare_13 : Bool;   // System status - Spare
         Ax1_PositionedRight : Bool;   // System status - Motor 1 Section 1 - positioned on the right
         Ax1_PositionedLeft : Bool;   // System status - Motor 1 Section 1 - positioned on the left
      END_STRUCT;
      "FromMCAx[1]" : Struct   // Axis 1 status word
         Fwd_Running : Bool;   // Axis selected status - Motor in forward running
         Bkwd_Running : Bool;   // Axis selected status - Motor in backward running
         Aborted : Bool;   // Axis selected status - current procedure or command aborted
         STO_Ok : Bool;   // Axis selected status - Safe torque OFF ok
         Fault : Bool;   // Axis selected status - Fault
         Bypass : Bool;   // Axis selected status - Axis bypassed
         Spare_6 : Bool;   // Axis selected status - Spare
         ZeroDone : Bool;   // Axis selected status - 0 performed on actual position
         Ready : Bool;   // Axis selected status - ready for operation
         Servo_active : Bool;   // Axis selected status - servo mode active
         Homing : Bool;   // Axis selected status - homing procedure in progress
         Homed : Bool;   // Axis selected status - homing performed
         Positioning : Bool;   // Axis selected status - positioning in progress
         Positioned : Bool;   // Axis selected status - positioned
         Standstill : Bool;   // Axis selected status - motor stopped
         Spare_15 : Bool;   // Axis selected status - Spare
      END_STRUCT;
      "FromMCAx[1]ErrorCode" : Int;   // Axis 1 status - Error code
      "FromMCAx[1]ActualSpeed" : Int;   // Axis 1 status - Actual speed [degrees*10/s]
      "FromMCAx[1]ActualCurrent" : Int;   // Axis 1 status - Actual current [A*100]
      "FromMCAx[1]ActualTorque" : Int;   // Axis 1 status - Actual torque [%*100]
      "FromMCAx[1]ActualPosition" : Int;   // Axis 1 status - Actual position [degrees*100]
      "FromMCAx[2]" : Struct   // Axis 2 status word
         Fwd_Running : Bool;   // Axis selected status - Motor in forward running
         Bkwd_Running : Bool;   // Axis selected status - Motor in backward running
         Aborted : Bool;   // Axis selected status - current procedure or command aborted
         STO_Ok : Bool;   // Axis selected status - Safe torque OFF ok
         Fault : Bool;   // Axis selected status - Fault
         Spare_5 : Bool;   // Axis selected status - Spare
         Spare_6 : Bool;   // Axis selected status - Spare
         ZeroDone : Bool;   // Axis selected status - 0 performed on actual position
         Ready : Bool;   // Axis selected status - ready for operation
         Servo_active : Bool;   // Axis selected status - servo mode active
         Homing : Bool;   // Axis selected status - homing procedure in progress
         Homed : Bool;   // Axis selected status - homing performed
         Positioning : Bool;   // Axis selected status - positioning in progress
         Positioned : Bool;   // Axis selected status - positioned
         Standstill : Bool;   // Axis selected status - motor stopped
         Spare_15 : Bool;   // Axis selected status - Spare
      END_STRUCT;
      "FromMCAx[2]ErrorCode" : Int;   // Axis 2 status - Error code
      "FromMCAx[2]ActualSpeed" : Int;   // Axis 2 status - Actual speed [mm/s*10]
      "FromMCAx[2]ActualCurrent" : Int;   // Axis 2 status - Actual current [A*100]
      "FromMCAx[2]ActualTorque" : Int;   // Axis 2 status - Actual torque [%*100]
      "FromMCAx[2]ActualPosition" : Int;   // Axis 2 status - Actual position [degrees*100]
   END_STRUCT;

END_TYPE

TYPE "UDT_VfdKebaSystemConfiguration"
VERSION : 0.1
   STRUCT
      VFDPNDeviceName : String;   // VFD's device name
      PositioningAxis { S7_SetPoint := 'False'} : "UDT_VfdKebaSystemPositioningAxisConfiguration";   // Positioning axis configuration
      SpeedAxis { S7_SetPoint := 'False'} : "UDT_VfdKebaSystemSpeedAxisConfiguration";   // Speed axis configuration
   END_STRUCT;

END_TYPE

FUNCTION_BLOCK "FB_VfdKebaSystem"
TITLE = FB_VFD_SEW_MOVI-C_Positioning
{ S7_Optimized_Access := 'TRUE' }
AUTHOR : MHSE
VERSION : 3.0
// ATTRIBUTES
// AUTO_NUMBER = True
// BLOCK_NUMBER = 86
// END_ATTRIBUTES
//Control SEW Servo VFD with multiple positions
   VAR_INPUT
      iUDT_VFDConfiguration { ExternalAccessible := 'False'; ExternalVisible := 'False'; ExternalWritable := 'False'} : "UDT_VfdKebaSystemConfiguration";   // Configuration structure
      iUDT_VFDInputs { ExternalAccessible := 'False'; ExternalVisible := 'False'; ExternalWritable := 'False'} : "UDT_VfdKebaSystemPI";   // VFD inputs structure
      ix_MainPowerOk { ExternalAccessible := 'False'; ExternalVisible := 'False'; ExternalWritable := 'False'} : Bool;   // TRUE when main power is ok
      ix_SimulationModeActive { ExternalAccessible := 'False'; ExternalVisible := 'False'; ExternalWritable := 'False'} : Bool;   // Simulation On
      ix_SafetyReset { ExternalAccessible := 'False'; ExternalVisible := 'False'; ExternalWritable := 'False'} : Bool;   // Safety reset
   END_VAR

   VAR_OUTPUT
      qUDT_HMIStatus { ExternalAccessible := 'False'; ExternalVisible := 'False'; ExternalWritable := 'False'} : "UDT_VfdKebaSystemStatus";   // HMI status structure
      qUDT_VFDOutputs { ExternalAccessible := 'False'; ExternalVisible := 'False'; ExternalWritable := 'False'} : "UDT_VfdKebaSystemPO";   // VFD outputs structure
   END_VAR

   VAR_IN_OUT
      iqUDT_PolisorterInterface : "UDT_PolisorterInterface";   // Polisorter interface structure
      iqUDT_ConveyorInterface : "UDT_ConveyorInterface";   // Polisorter conveyor interface structure
      iqUDT_VFDStatistics : "UDT_VfdKebaSystemStatistics";   // VFD statistics
   END_VAR

   VAR
      sUDT_PNDevice { ExternalAccessible := 'False'; ExternalVisible := 'False'; ExternalWritable := 'False'; S7_SetPoint := 'False'} : "UDT_PNDevice";   //  PN device info structure
      sUDT_HMIStatus { ExternalAccessible := 'False'; ExternalVisible := 'False'; ExternalWritable := 'False'; S7_SetPoint := 'False'} : "UDT_VfdKebaSystemStatus";   // Status struture
      sa_PNPortsStatus { ExternalAccessible := 'False'; ExternalVisible := 'False'; ExternalWritable := 'False'} : Array[1..8] of Bool;   // TRUE when specific port has an error
      sFB_TimerOnOffDelayCheckSupply { ExternalAccessible := 'False'; ExternalVisible := 'False'; ExternalWritable := 'False'; S7_SetPoint := 'False'} : "FB_TimerOnOffDelay";   // MHS "TimerOnOffDelay" - to delay time for VFD supply contactor
      sFB_TimerOnOffDelayAliveCount { ExternalAccessible := 'False'; ExternalVisible := 'False'; ExternalWritable := 'False'; S7_SetPoint := 'False'} : "FB_TimerOnOffDelay";   // MHS "TimerOnOffDelay" - to delay time for communication feedback
      sFB_TimerOnOffDelayPositioning { ExternalAccessible := 'False'; ExternalVisible := 'False'; ExternalWritable := 'False'; S7_SetPoint := 'False'} : "FB_TimerOnOffDelay";   // MHS "TimerOnOffDelay" - to delay time for positioning error
      sFB_TimerOnOffDelay_PostionRequestDelay { ExternalAccessible := 'False'; ExternalVisible := 'False'; ExternalWritable := 'False'; S7_SetPoint := 'False'} : "FB_TimerOnOffDelay";   // MHS "TimerOnOffDelay" - to delay time for position request
      sFB_TimerOnOffDelay_SafetyResetPulse { ExternalAccessible := 'False'; ExternalVisible := 'False'; ExternalWritable := 'False'; S7_SetPoint := 'False'} : "FB_TimerOnOffDelay";   // MHS "TimerOnOffDelay" - to delay time for safety reset
      sFB_TimerOnOffDelay_Reset { ExternalAccessible := 'False'; ExternalVisible := 'False'; ExternalWritable := 'False'; S7_SetPoint := 'False'} : "FB_TimerOnOffDelay";   // MHS "TimerOnOffDelay" - to delay time for reset
      sF_TRIG_LST {InstructionName := 'F_TRIG'; LibVersion := '1.0'; ExternalAccessible := 'False'; ExternalVisible := 'False'; ExternalWritable := 'False'; S7_SetPoint := 'False'} : F_TRIG;   // Falling edge positioning feedback
      sR_TRIG_ManInPos {InstructionName := 'R_TRIG'; LibVersion := '1.0'; ExternalAccessible := 'False'; ExternalVisible := 'False'; ExternalWritable := 'False'; S7_SetPoint := 'False'} : R_TRIG;   // Rising edge manual travel into position
      sR_TRIG_PNSlaveNotOnline {InstructionName := 'R_TRIG'; LibVersion := '1.0'; ExternalAccessible := 'False'; ExternalVisible := 'False'; ExternalWritable := 'False'; S7_SetPoint := 'False'} : R_TRIG;   // Rising edge for trigger Profinet slave not online statistics
      sR_TRIG_PNSlaveError {InstructionName := 'R_TRIG'; LibVersion := '1.0'; ExternalAccessible := 'False'; ExternalVisible := 'False'; ExternalWritable := 'False'; S7_SetPoint := 'False'} : R_TRIG;   // Rising edge for trigger Profinet slave error statistics
      sR_TRIG_Ax1_InternalError {InstructionName := 'R_TRIG'; LibVersion := '1.0'; ExternalAccessible := 'False'; ExternalVisible := 'False'; ExternalWritable := 'False'; S7_SetPoint := 'False'} : R_TRIG;   // Rising edge for trigger axis 1 Internal VFD Error statistics
      sR_TRIG_Ax2_InternalError {InstructionName := 'R_TRIG'; LibVersion := '1.0'; ExternalAccessible := 'False'; ExternalVisible := 'False'; ExternalWritable := 'False'; S7_SetPoint := 'False'} : R_TRIG;   // Rising edge for trigger axis 2 Internal VFD Error statistics
      sR_TRIG_CommunicationError {InstructionName := 'R_TRIG'; LibVersion := '1.0'; ExternalAccessible := 'False'; ExternalVisible := 'False'; ExternalWritable := 'False'; S7_SetPoint := 'False'} : R_TRIG;   // Rising edge for trigger communication error statistics
      sR_TRIG_Ax1_Running {InstructionName := 'R_TRIG'; LibVersion := '1.0'; ExternalAccessible := 'False'; ExternalVisible := 'False'; ExternalWritable := 'False'; S7_SetPoint := 'False'} : R_TRIG;   // Rising edge for starting of the axis 1 running signal
      sR_TRIG_Ax2_Running {InstructionName := 'R_TRIG'; LibVersion := '1.0'; ExternalAccessible := 'False'; ExternalVisible := 'False'; ExternalWritable := 'False'; S7_SetPoint := 'False'} : R_TRIG;   // Rising edge for starting of the axis 2 running signal
      sr_Ax1ActualCurrent { ExternalAccessible := 'False'; ExternalVisible := 'False'; ExternalWritable := 'False'} : Real;   // Axis 1 actual current [A]
      sr_Ax1ActualTorque { ExternalAccessible := 'False'; ExternalVisible := 'False'; ExternalWritable := 'False'} : Real;   // Axis 1 actual torque [Nm]
      sr_Ax2ActualCurrent { ExternalAccessible := 'False'; ExternalVisible := 'False'; ExternalWritable := 'False'} : Real;   // Axis 2 actual current [A]
      sr_Ax2ActualTorque { ExternalAccessible := 'False'; ExternalVisible := 'False'; ExternalWritable := 'False'} : Real;   // Axis 2 actual torque [Nm]
      sdi_ActualPositionValue { ExternalAccessible := 'False'; ExternalVisible := 'False'; ExternalWritable := 'False'} : DInt;   // Axis 1 actual position [degree]
      sr_Ax1ActualSpeed { ExternalAccessible := 'False'; ExternalVisible := 'False'; ExternalWritable := 'False'} : Int;   // Axis 1 actual speed  [degree/s]
      sr_Ax2ActualSpeed { ExternalAccessible := 'False'; ExternalVisible := 'False'; ExternalWritable := 'False'} : Int;   // Axis 2 actual speed  [mm/s]
      si_LastSwitchtime { ExternalAccessible := 'False'; ExternalVisible := 'False'; ExternalWritable := 'False'} : Int;   // The actual time it took the last switch-over
      si_AliveCountToKEBA { ExternalAccessible := 'False'; ExternalVisible := 'False'; ExternalWritable := 'False'} : Int;
      si_OldSpeed { ExternalAccessible := 'False'; ExternalVisible := 'False'; ExternalWritable := 'False'} : Int;   // Old speed setpoint for manual mode speed change during movement
      si_AliveCount { ExternalAccessible := 'False'; ExternalVisible := 'False'; ExternalWritable := 'False'} : Int;   //  Handshake to movikit
      sx_Ax1_ErrorActive { ExternalAccessible := 'False'; ExternalVisible := 'False'; ExternalWritable := 'False'} : Bool;   // Axis 1 error active
      sx_Ax2_ErrorActive { ExternalAccessible := 'False'; ExternalVisible := 'False'; ExternalWritable := 'False'} : Bool;   // Axis 2 error active
      sx_Ax1_WarningActive { ExternalAccessible := 'False'; ExternalVisible := 'False'; ExternalWritable := 'False'} : Bool;   // Axis 1 warning active
      sx_PNDeviceHealthy { ExternalAccessible := 'False'; ExternalVisible := 'False'; ExternalWritable := 'False'} : Bool;   // PN Device is healthy, no errors
      sx_AliveCountFeedback { ExternalAccessible := 'False'; ExternalVisible := 'False'; ExternalWritable := 'False'} : Bool;   //  Movikit feedback delay
      sx_HardwareAvailable { ExternalAccessible := 'False'; ExternalVisible := 'False'; ExternalWritable := 'False'} : Bool;   // All hardware is on line and available
      sx_PowerOK { ExternalAccessible := 'False'; ExternalVisible := 'False'; ExternalWritable := 'False'} : Bool;   // All Power (in and external) is ok
      sx_PositioningFeedback { ExternalAccessible := 'False'; ExternalVisible := 'False'; ExternalWritable := 'False'} : Bool;   // Positioning feedback delay
      sx_Ax1_Ready { ExternalAccessible := 'False'; ExternalVisible := 'False'; ExternalWritable := 'False'} : Bool;   // Axis 1 control is ready to operate
      sx_Ax2_Ready { ExternalAccessible := 'False'; ExternalVisible := 'False'; ExternalWritable := 'False'} : Bool;   // Axis 2 control is ready to operate
      sx_ManualPositionStop { ExternalAccessible := 'False'; ExternalVisible := 'False'; ExternalWritable := 'False'} : Bool;   // A configured position is reached in manual mode
      sx_ManualPosHold { ExternalAccessible := 'False'; ExternalVisible := 'False'; ExternalWritable := 'False'} : Bool;   // Hold in position
      sx_ConfigurationError { ExternalAccessible := 'False'; ExternalVisible := 'False'; ExternalWritable := 'False'} : Bool;   // Commissioning: configuration of parameters is wrong
      sx_ResetPulse { ExternalAccessible := 'False'; ExternalVisible := 'False'; ExternalWritable := 'False'} : Bool;   // Reset pulse
      sx_SpeedChange { ExternalAccessible := 'False'; ExternalVisible := 'False'; ExternalWritable := 'False'} : Bool;   // Speed change for manual mode speed change during movement
   END_VAR

   VAR CONSTANT
      ci_NumberOfProfinetPorts : Int := 2;   // Number of Profinet ports in device
      ci_NoMode : Int := 0;   // Operation mode: No mode
      ci_AutoMode : Int := 1;   // Operation mode: Auto mode
      ci_ManualMode : Int := 2;   // Operation mode: Manual mode
      ci_Maintenance : Int := 10;   // Operation mode: Maintenace mode
      ci_MaintenanceManualMode : Int := 12;   // Operation mode: Maintenace manual mode
      ci_MaintenanceHoming : Int := 13;   // Operation mode: Maintenace homing mode
      ci_MaintenanceStressTest : Int := 14;   // Operation mode: Maintenace stress test  mode
      ci_RotationManualSpeedLinit : Int := 12;   // Rotation speed limit for manual mode
   END_VAR


BEGIN
	(*
	----------------------------------------------------------------------------------------

	Version history:
	Date        | Version   | Author        | Remark
	----------------------------------------------------------------------------------------
	26/10/2021  | 0.1       | L.Klar        | first release MHS TIA 16
	21/02/2023  | 4.0       | F.Baten       | 4.0 Release TIA 17.5
	*)

	REGION 1 - Get Device Profinet information

	    "FC_GetDevicePN"(is_PNDeviceName := #iUDT_VFDConfiguration.VFDPNDeviceName,
	                     ix_SimulationModeActive := #ix_SimulationModeActive,
	                     iqUDT_PND := #sUDT_PNDevice);


	    "FC_GetPNPortStatus"(ii_NumberOfPorts := #ci_NumberOfProfinetPorts,
	                         iUDT_DevicePNInfo := #sUDT_PNDevice,
	                         qa_PortFault => #sa_PNPortsStatus);

	END_REGION

	REGION 2 - Reset errors

	    // Reset pulse
	    #sFB_TimerOnOffDelay_Reset(iudi_OffDelayTime := 200,
	                               ix_SignalToDelay := #iqUDT_PolisorterInterface.InternalErrorReset OR #iqUDT_ConveyorInterface.InternalErrorReset,
	                               qx_DelayedSignal => #sx_ResetPulse);

	    // Internal errors reset
	    IF #sx_ResetPulse

	    THEN
	        #sUDT_HMIStatus.PNSlaveNotOnline := FALSE;
	        #sUDT_HMIStatus.PNSlaveError := FALSE;
	        #sUDT_HMIStatus.PositioningTimeWarning := FALSE;
	        #sUDT_HMIStatus.Axis1InternalError := FALSE;
	        #sUDT_HMIStatus.PNSlaveWarning := FALSE;
	        #sUDT_HMIStatus.CommunicationError := FALSE;

	    END_IF;

	    // KEBA reset outputs
	    #qUDT_VFDOutputs.ToMCControl1.Reset := #sx_ResetPulse;
	    #qUDT_VFDOutputs."ToMCAx[1]".Reset := #sx_ResetPulse;
	    #qUDT_VFDOutputs."ToMCAx[2]".Reset := #sx_ResetPulse;

	    // Safety reset pulse
	    #sFB_TimerOnOffDelay_SafetyResetPulse(iudi_OffDelayTime := 100,
	                                          ix_SignalToDelay := #ix_SafetyReset,
	                                          qx_DelayedSignal => #qUDT_VFDOutputs.ToMCControl1.LocalSafetyReset);

	END_REGION

	REGION 3 - Check Hardware

	    REGION 3.1 - Power OK
	        // Hardware will be available after delay so the device has time for initialisation
	        #sFB_TimerOnOffDelayCheckSupply(iudi_OnDelayTime := 2000,
	                                        ix_SignalToDelay := #ix_MainPowerOk);

	        #sx_PowerOK := #sFB_TimerOnOffDelayCheckSupply.qx_DelayedSignal;
	    END_REGION

	    REGION 3.2 - PN Healthy Check

	        IF NOT "DB_ProfinetDiagnostic".ProfinetNetworks[#sUDT_PNDevice.PNNetworknumber].DeviceStatus[#sUDT_PNDevice.PNDeviceNumber].DeviceState.Exist
	            AND NOT #ix_SimulationModeActive
	            AND #sx_PowerOK
	        THEN
	            #sUDT_HMIStatus.PNSlaveNotOnline := TRUE;
	        END_IF;

	        // Check if PN ports are healthy
	        IF #sa_PNPortsStatus[1] XOR #sa_PNPortsStatus[2] THEN
	            #sUDT_HMIStatus.PNSlaveWarning := TRUE;
	        END_IF;

	        IF "DB_ProfinetDiagnostic".ProfinetNetworks[#sUDT_PNDevice.PNNetworknumber].DeviceStatus[#sUDT_PNDevice.PNDeviceNumber].DeviceState.Error
	            AND NOT #ix_SimulationModeActive
	            AND #sx_PowerOK
	            AND NOT #sUDT_HMIStatus.PNSlaveWarning

	        THEN
	            #sUDT_HMIStatus.PNSlaveError := TRUE;
	        END_IF;

	        #sx_PNDeviceHealthy := NOT #sUDT_HMIStatus.PNSlaveNotOnline
	        AND NOT #sUDT_HMIStatus.PNSlaveError
	        AND #sx_PowerOK
	        AND #sUDT_PNDevice.PNDeviceFound;

	    END_REGION

	    REGION 3.3 - Hardware is available

	        #sx_HardwareAvailable := #sx_PowerOK
	        AND #sx_PNDeviceHealthy
	        OR #ix_SimulationModeActive;

	    END_REGION

	    REGION 3.4 - Check communication Alive Count

	        // Alive count check
	        #sx_AliveCountFeedback := #si_AliveCount = #iUDT_VFDInputs.FromMCAliveCount;

	        #sFB_TimerOnOffDelayAliveCount(iudi_OnDelayTime := 2000,
	                                       ix_SignalToDelay := #sx_AliveCountFeedback);

	        IF (#sFB_TimerOnOffDelayAliveCount.qx_DelayedSignal)
	            AND #sx_HardwareAvailable
	        THEN
	            #sUDT_HMIStatus.CommunicationError := TRUE;
	        END_IF;

	        #si_AliveCount := #iUDT_VFDInputs.FromMCAliveCount;

	        // Alive count for KEBA
	        IF "DB_Memory"."OS_0.1sec"
	        THEN
	            #qUDT_VFDOutputs.ToMCAliveCount := #si_AliveCountToKEBA;
	            #si_AliveCountToKEBA += 1;

	            IF #si_AliveCountToKEBA > 9999
	            THEN
	                #si_AliveCountToKEBA := 0;
	            END_IF;
	        END_IF;

	    END_REGION

	END_REGION

	REGION 4 - Handle input data

	    REGION 4.1 - Move to status

	        // Axis 1
	        #sr_Ax1ActualTorque := INT_TO_REAL(#iUDT_VFDInputs."FromMCAx[1]ActualTorque" / 100);
	        #sr_Ax1ActualCurrent := INT_TO_REAL(#iUDT_VFDInputs."FromMCAx[1]ActualCurrent" / 100);
	        #sr_Ax1ActualSpeed := #iUDT_VFDInputs."FromMCAx[1]ActualSpeed" / 10;

	        // Axis 2
	        #sr_Ax2ActualTorque := INT_TO_REAL(#iUDT_VFDInputs."FromMCAx[2]ActualTorque" / 100);
	        #sr_Ax2ActualCurrent := INT_TO_REAL(#iUDT_VFDInputs."FromMCAx[2]ActualCurrent" / 100);
	        #sr_Ax2ActualSpeed := #iUDT_VFDInputs."FromMCAx[2]ActualSpeed" / 10;

	    END_REGION

	    REGION 4.2 - Actual positon value

	        #sdi_ActualPositionValue := #iUDT_VFDInputs."FromMCAx[1]ActualPosition" / 100;

	        IF #sdi_ActualPositionValue <= (#iUDT_VFDConfiguration.PositioningAxis.Position[#iqUDT_PolisorterInterface.PositionSetpoint] + #iUDT_VFDConfiguration.PositioningAxis.PositionWindow)
	            AND #sdi_ActualPositionValue >= (#iUDT_VFDConfiguration.PositioningAxis.Position[#iqUDT_PolisorterInterface.PositionSetpoint] - #iUDT_VFDConfiguration.PositioningAxis.PositionWindow)

	        THEN
	            #iqUDT_PolisorterInterface.PositionActual := #iqUDT_PolisorterInterface.PositionSetpoint;
	        ELSE
	            #iqUDT_PolisorterInterface.PositionActual := 0;
	        END_IF;

	    END_REGION

	    REGION 4.3 - Manual position

	        // Logic to stop at a predefined position when jogging. After the stop, the movement can restarted by pressing the jog button again
	        IF #iUDT_VFDInputs.FromMCActiveOpMode = #ci_ManualMode
	        THEN
	            #sx_ManualPositionStop :=
	            (#sdi_ActualPositionValue <= (#iUDT_VFDConfiguration.PositioningAxis.Position[1] + #iUDT_VFDConfiguration.PositioningAxis.PositionWindow)
	            AND #sdi_ActualPositionValue >= (#iUDT_VFDConfiguration.PositioningAxis.Position[1] - #iUDT_VFDConfiguration.PositioningAxis.PositionWindow))
	            OR (#sdi_ActualPositionValue <= (#iUDT_VFDConfiguration.PositioningAxis.Position[2] + #iUDT_VFDConfiguration.PositioningAxis.PositionWindow)
	            AND #sdi_ActualPositionValue >= (#iUDT_VFDConfiguration.PositioningAxis.Position[2] - #iUDT_VFDConfiguration.PositioningAxis.PositionWindow))
	            OR (#sdi_ActualPositionValue <= (#iUDT_VFDConfiguration.PositioningAxis.Position[3] + #iUDT_VFDConfiguration.PositioningAxis.PositionWindow)
	            AND #sdi_ActualPositionValue >= (#iUDT_VFDConfiguration.PositioningAxis.Position[3] - #iUDT_VFDConfiguration.PositioningAxis.PositionWindow))
	            OR (#sdi_ActualPositionValue <= (#iUDT_VFDConfiguration.PositioningAxis.Position[4] + #iUDT_VFDConfiguration.PositioningAxis.PositionWindow)
	            AND #sdi_ActualPositionValue >= (#iUDT_VFDConfiguration.PositioningAxis.Position[4] - #iUDT_VFDConfiguration.PositioningAxis.PositionWindow))
	            OR (#sdi_ActualPositionValue <= (#iUDT_VFDConfiguration.PositioningAxis.Position[5] + #iUDT_VFDConfiguration.PositioningAxis.PositionWindow)
	            AND #sdi_ActualPositionValue >= (#iUDT_VFDConfiguration.PositioningAxis.Position[5] - #iUDT_VFDConfiguration.PositioningAxis.PositionWindow))
	            OR (#sdi_ActualPositionValue <= (#iUDT_VFDConfiguration.PositioningAxis.Position[6] + #iUDT_VFDConfiguration.PositioningAxis.PositionWindow)
	            AND #sdi_ActualPositionValue >= (#iUDT_VFDConfiguration.PositioningAxis.Position[6] - #iUDT_VFDConfiguration.PositioningAxis.PositionWindow))
	            OR (#sdi_ActualPositionValue <= (#iUDT_VFDConfiguration.PositioningAxis.Position[7] + #iUDT_VFDConfiguration.PositioningAxis.PositionWindow)
	            AND #sdi_ActualPositionValue >= (#iUDT_VFDConfiguration.PositioningAxis.Position[7] - #iUDT_VFDConfiguration.PositioningAxis.PositionWindow))
	            OR (#sdi_ActualPositionValue <= (#iUDT_VFDConfiguration.PositioningAxis.Position[8] + #iUDT_VFDConfiguration.PositioningAxis.PositionWindow)
	            AND #sdi_ActualPositionValue >= (#iUDT_VFDConfiguration.PositioningAxis.Position[8] - #iUDT_VFDConfiguration.PositioningAxis.PositionWindow))
	            OR (#sdi_ActualPositionValue <= (#iUDT_VFDConfiguration.PositioningAxis.Position[9] + #iUDT_VFDConfiguration.PositioningAxis.PositionWindow)
	            AND #sdi_ActualPositionValue >= (#iUDT_VFDConfiguration.PositioningAxis.Position[9] - #iUDT_VFDConfiguration.PositioningAxis.PositionWindow))
	            OR (#sdi_ActualPositionValue <= (#iUDT_VFDConfiguration.PositioningAxis.Position[10] + #iUDT_VFDConfiguration.PositioningAxis.PositionWindow)
	            AND #sdi_ActualPositionValue >= (#iUDT_VFDConfiguration.PositioningAxis.Position[10] - #iUDT_VFDConfiguration.PositioningAxis.PositionWindow));
	        END_IF;

	    END_REGION

	END_REGION

	REGION 5 - Errors and warnings

	    REGION 5.1 - VFD internal error

	        // Axis 1
	        #sUDT_HMIStatus.Axis1InternalError := #iUDT_VFDInputs."FromMCAx[1]".Fault;
	        #sUDT_HMIStatus.AX1ErrorCode := #iUDT_VFDInputs."FromMCAx[1]ErrorCode";

	        IF NOT #iUDT_VFDInputs."FromMCAx[1]".Fault
	        THEN
	            #sUDT_HMIStatus.AX1ErrorCode := 0;
	        END_IF;

	        // Axis 2
	        #sUDT_HMIStatus.Axis2InternalError := #iUDT_VFDInputs."FromMCAx[2]".Fault;
	        #sUDT_HMIStatus.AX2ErrorCode := #iUDT_VFDInputs."FromMCAx[2]ErrorCode";

	        IF NOT #iUDT_VFDInputs."FromMCAx[2]".Fault
	        THEN
	            #sUDT_HMIStatus.AX2ErrorCode := 0;
	        END_IF;

	    END_REGION

	    REGION 5.2 - Positioning warning

	        // This timer checks if the speed of the VFD is ok.
	        // The VFD should reach is next destination in the given time

	        #sx_PositioningFeedback := #iqUDT_PolisorterInterface.PositionActual <> #iqUDT_PolisorterInterface.PositionSetpoint
	        AND #iqUDT_PolisorterInterface.Automatic;

	        #sF_TRIG_LST(CLK := #sx_PositioningFeedback);

	        IF #sF_TRIG_LST.Q
	        THEN
	            #si_LastSwitchtime := LREAL_TO_INT(#sFB_TimerOnOffDelayPositioning.qlr_ActualTime);
	        END_IF;

	        #sFB_TimerOnOffDelayPositioning(iudi_OnDelayTime := (#iqUDT_PolisorterInterface.SwitchingTime + 100),
	                                        ix_SignalToDelay := #sx_PositioningFeedback);

	        IF #sFB_TimerOnOffDelayPositioning.qx_DelayedSignal
	        THEN
	            #sUDT_HMIStatus.PositioningTimeWarning := TRUE;
	        END_IF;

	    END_REGION

	    REGION 5.3 - Common Error

	        // Axis 1 VFD error active
	        #sx_Ax1_ErrorActive := #sUDT_HMIStatus.Axis1InternalError
	        OR #sUDT_HMIStatus.CommunicationError;

	        // Axis 1 VFD error active
	        #sx_Ax2_ErrorActive := #sUDT_HMIStatus.Axis2InternalError
	        OR #sUDT_HMIStatus.CommunicationError;

	    END_REGION

	    REGION 5.4 - Configuration Error

	        //  Check if no faulty setup is active
	        //  This is the responcebility of the commisioning engineer
	        IF #iUDT_VFDConfiguration.PositioningAxis.PositionMax > #iUDT_VFDConfiguration.PositioningAxis.PositionMin
	            AND #iUDT_VFDConfiguration.PositioningAxis.PositionMax > 0
	            AND #iUDT_VFDConfiguration.PositioningAxis.VFDSpeed > 0
	            AND #iUDT_VFDConfiguration.SpeedAxis.Acceleration > 0
	            AND #iUDT_VFDConfiguration.SpeedAxis.Deceleration > 0
	            AND "DB_ProfinetDiagnostic".ProfinetNetworks[#sUDT_PNDevice.PNNetworknumber].DeviceStatus[#sUDT_PNDevice.PNDeviceNumber].DeviceState.Configure
	        THEN
	            #sx_ConfigurationError := FALSE;
	        ELSE
	            #sx_ConfigurationError := TRUE;
	        END_IF;

	    END_REGION

	    REGION 5.5 - Common warning

	        // Set VFD warning active
	        #sx_Ax1_WarningActive := #sUDT_HMIStatus.PositioningTimeWarning;

	    END_REGION

	END_REGION

	REGION 6 - Check conditions to set VFD Ready signals

	    REGION 6.1 - Internal VFD ready

	        // Axis 1
	        #sx_Ax1_Ready := #sx_HardwareAvailable
	        AND (#iUDT_VFDInputs."FromMCAx[1]".Ready
	        OR #iUDT_VFDInputs.FromMCStatus1.Running)
	        AND NOT #sx_Ax1_ErrorActive
	        AND NOT #sx_ConfigurationError
	        AND (#iUDT_VFDInputs."FromMCAx[1]".STO_Ok OR #iUDT_VFDInputs."FromMCAx[1]".Bypass);

	        // Axis 2
	        #sx_Ax2_Ready := #sx_HardwareAvailable
	        AND (#iUDT_VFDInputs."FromMCAx[2]".Ready
	        OR #iUDT_VFDInputs.FromMCStatus1.Running)
	        AND NOT #sx_Ax1_ErrorActive
	        AND NOT #sx_ConfigurationError
	        AND #iUDT_VFDInputs."FromMCAx[2]".STO_Ok;

	    END_REGION

	    REGION 6.2 - External VFD ready (to control)

	        #iqUDT_PolisorterInterface.Ready :=
	        (#iqUDT_PolisorterInterface.Automatic
	        AND NOT #iqUDT_PolisorterInterface.Manual
	        AND #iUDT_VFDInputs.FromMCStatus1.Homed
	        AND #iUDT_VFDInputs.FromMCActiveOpMode = #ci_AutoMode)
	        OR
	        (NOT #iqUDT_PolisorterInterface.Automatic
	        AND #iqUDT_PolisorterInterface.Manual
	        AND #iUDT_VFDInputs.FromMCActiveOpMode = #ci_ManualMode)
	        AND
	        #iqUDT_PolisorterInterface.RunEnabled;

	    END_REGION

	END_REGION

	REGION 7 - Set VFD control data

	    REGION 7.1 - Initialize variables

	        // Operating mode
	        #qUDT_VFDOutputs.ToMCActiveOpMode := #ci_NoMode;

	        // Axis 1
	        #qUDT_VFDOutputs."ToMCAx[1]SpeedSetpoint" := 0;
	        #qUDT_VFDOutputs.ToMCControl1.ServoON := FALSE;
	        #qUDT_VFDOutputs.ToMCControl1.Start := FALSE;

	        #qUDT_VFDOutputs."ToMCAx[1]".Servo_ON := FALSE;
	        #qUDT_VFDOutputs."ToMCAx[1]".Jog_Fwd := FALSE;
	        #qUDT_VFDOutputs."ToMCAx[1]".Jog_Bkwd := FALSE;

	        // Axis 2
	        #qUDT_VFDOutputs."ToMCAx[2]".Servo_ON := FALSE;
	        #qUDT_VFDOutputs.ToMCControl2.Ax_BeltRunFwd := FALSE;
	        #qUDT_VFDOutputs.ToMCControl2.Ax_BeltRunBkwd := FALSE;
	        #qUDT_VFDOutputs."ToMCAx[2]SpeedSetpoint" := 0;

	        #qUDT_VFDOutputs."ToMCAx[2]".Servo_ON := FALSE;
	        #qUDT_VFDOutputs."ToMCAx[2]".Jog_Fwd := FALSE;
	        #qUDT_VFDOutputs."ToMCAx[2]".Jog_Bkwd := FALSE;

	        #qUDT_VFDOutputs."ToMCAx[2]SpeedSetpoint" := 0;
	        #qUDT_VFDOutputs."ToMCAx[2]Acceleration" := 0;
	        #qUDT_VFDOutputs."ToMCAx[2]Deceleration" := 0;

	    END_REGION

	    REGION 7.2 - Manual mode - jogging

	        IF #sx_Ax1_Ready
	            AND #iqUDT_PolisorterInterface.Manual
	            AND NOT #iqUDT_PolisorterInterface.Automatic
	            AND #iqUDT_PolisorterInterface.RunEnabled
	            AND NOT #iUDT_VFDInputs."FromMCAx[1]".Bypass

	        THEN

	            // Speed setpoint (saturated to 12 degree/s)
	            IF #iUDT_VFDConfiguration.PositioningAxis.VFDSpeed > #ci_RotationManualSpeedLinit THEN
	                #qUDT_VFDOutputs."ToMCAx[1]SpeedSetpoint" := 12 * 10;
	            ELSE
	                #qUDT_VFDOutputs."ToMCAx[1]SpeedSetpoint" := #iUDT_VFDConfiguration.PositioningAxis.VFDSpeed * 10;
	            END_IF;

	            #qUDT_VFDOutputs.ToMCActiveOpMode := #ci_ManualMode;

	            // Servo On
	            #qUDT_VFDOutputs."ToMCAx[1]".Servo_ON := #iUDT_VFDInputs.FromMCActiveOpMode = #ci_ManualMode
	            AND #iUDT_VFDInputs."FromMCAx[1]".Ready;

	            // Manual commands
	            IF #iUDT_VFDInputs.FromMCActiveOpMode = #ci_ManualMode
	                AND #iUDT_VFDInputs."FromMCAx[1]".Servo_active
	            THEN

	                // On position while jogging: stop, when button is released and pressed again continue to travel
	                #sR_TRIG_ManInPos(CLK := #sx_ManualPositionStop);

	                #sx_ManualPosHold := (#sx_ManualPosHold
	                OR #sR_TRIG_ManInPos.Q)
	                AND (#iqUDT_PolisorterInterface.JogLeft
	                OR #iqUDT_PolisorterInterface.JogRight)
	                AND #iqUDT_PolisorterInterface.Ready;

	                // Jog commands

	                IF #iqUDT_PolisorterInterface.Ready
	                    AND #iqUDT_PolisorterInterface.JogLeft
	                    AND NOT #iqUDT_PolisorterInterface.JogRight
	                    AND NOT #sx_ManualPosHold
	                THEN
	                    #qUDT_VFDOutputs."ToMCAx[1]".Jog_Fwd := TRUE;
	                    #qUDT_VFDOutputs."ToMCAx[1]".Jog_Bkwd := FALSE;
	                ELSIF
	                    #iqUDT_PolisorterInterface.Ready
	                    AND NOT #iqUDT_PolisorterInterface.JogLeft
	                    AND #iqUDT_PolisorterInterface.JogRight
	                    AND NOT #sx_ManualPosHold
	                THEN
	                    #qUDT_VFDOutputs."ToMCAx[1]".Jog_Fwd := FALSE;
	                    #qUDT_VFDOutputs."ToMCAx[1]".Jog_Bkwd := TRUE;
	                ELSE
	                    #qUDT_VFDOutputs."ToMCAx[1]".Jog_Fwd := FALSE;
	                    #qUDT_VFDOutputs."ToMCAx[1]".Jog_Bkwd := FALSE;

	                END_IF;

	            END_IF;

	        END_IF;

	    END_REGION

	    REGION 7.3 - Automatic mode - for positioning


	        IF #sx_Ax1_Ready
	            AND (#iUDT_VFDInputs."FromMCAx[1]".STO_Ok OR #iUDT_VFDInputs."FromMCAx[1]".Bypass)
	            AND #iqUDT_PolisorterInterface.Automatic
	            AND NOT #iqUDT_PolisorterInterface.Manual
	            AND #iqUDT_PolisorterInterface.RunEnabled
	            AND #iqUDT_PolisorterInterface.Referenced
	        THEN

	            // Auto mode start
	            #qUDT_VFDOutputs.ToMCActiveOpMode := #ci_AutoMode;

	            // Servo ON
	            #qUDT_VFDOutputs.ToMCControl1.ServoON := #iUDT_VFDInputs.FromMCActiveOpMode = #ci_AutoMode
	            AND #iUDT_VFDInputs."FromMCAx[1]".Ready;

	            // Servo is active
	            IF #iUDT_VFDInputs.FromMCStatus1.Servo_active AND NOT #iUDT_VFDInputs."FromMCAx[1]".Bypass
	            THEN

	                // Start auto mode
	                #qUDT_VFDOutputs.ToMCControl1.Start := TRUE;

	                // Speed setpoint
	                #qUDT_VFDOutputs."ToMCAx[1]SpeedSetpoint" := #iUDT_VFDConfiguration.PositioningAxis.VFDSpeed * 10;

	                // Initilialize positions setpoints
	                // #q_UDT_VFDOutputs."To_MC_Ax[1]PositionSetpointRight" := 0;
	                // #q_UDT_VFDOutputs."To_MC_Ax[1]PositionSetpointLeft" := 0;

	                // Position command delay
	                #sFB_TimerOnOffDelay_PostionRequestDelay(iudi_OnDelayTime := 100,
	                                                         ix_SignalToDelay := #iUDT_VFDInputs."FromMCAx[1]".Positioned AND #iUDT_VFDInputs."FromMCAx[1]".Standstill);

	                IF #sFB_TimerOnOffDelay_PostionRequestDelay.qx_DelayedSignal THEN
	                    // Position setpoint
	                    CASE #iqUDT_PolisorterInterface.PositionSetpoint OF
	                        1:
	                            #qUDT_VFDOutputs.ToMCControl2.Ax1_PosLeft := TRUE;
	                            #qUDT_VFDOutputs.ToMCControl2.Ax1_PosRight := FALSE;
	                            #qUDT_VFDOutputs."ToMCAx[1]PositionSetpointLeft" := #iUDT_VFDConfiguration.PositioningAxis.Position[#iqUDT_PolisorterInterface.PositionSetpoint] * 10;
	                            #qUDT_VFDOutputs."ToMCAx[1]PositionSetpointRight" := 0;
	                        2:
	                            #qUDT_VFDOutputs.ToMCControl2.Ax1_PosLeft := FALSE;
	                            #qUDT_VFDOutputs.ToMCControl2.Ax1_PosRight := FALSE;
	                            #qUDT_VFDOutputs."ToMCAx[1]PositionSetpointLeft" := 0;
	                            #qUDT_VFDOutputs."ToMCAx[1]PositionSetpointRight" := 0;
	                        3:
	                            #qUDT_VFDOutputs.ToMCControl2.Ax1_PosLeft := FALSE;
	                            #qUDT_VFDOutputs.ToMCControl2.Ax1_PosRight := TRUE;
	                            #qUDT_VFDOutputs."ToMCAx[1]PositionSetpointRight" := #iUDT_VFDConfiguration.PositioningAxis.Position[#iqUDT_PolisorterInterface.PositionSetpoint] * 10;
	                            #qUDT_VFDOutputs."ToMCAx[1]PositionSetpointLeft" := 0;
	                    END_CASE;
	                END_IF;
	            END_IF;
	        END_IF;

	    END_REGION

	    REGION 7.4 - Conveyor control

	        IF #sx_Ax2_Ready
	        THEN

	            // Speed change during manual mode (command needs to be reenabled to aplly new speed setpoint)
	            IF #iqUDT_ConveyorInterface.SpeedSetpoint <> #si_OldSpeed THEN
	                #si_OldSpeed := #iqUDT_ConveyorInterface.SpeedSetpoint;
	                #sx_SpeedChange := TRUE;
	            END_IF;

	            // Rotation direction
	            #qUDT_VFDOutputs."ToMCAx[2]".Direction := #iUDT_VFDConfiguration.SpeedAxis.DirectionReversal;
	            // Speed setpoint
	            #qUDT_VFDOutputs."ToMCAx[2]SpeedSetpoint" := #iqUDT_ConveyorInterface.SpeedSetpoint * 10;
	            // Speed correction
	            #qUDT_VFDOutputs."ToMCAx[2]Adjustment" := #iUDT_VFDConfiguration.SpeedAxis.BeltSpeedCorrection;

	            // Accelaeratio, deceleration
	            #qUDT_VFDOutputs."ToMCAx[2]Acceleration" := UINT_TO_INT(#iUDT_VFDConfiguration.SpeedAxis.Acceleration * 10);
	            #qUDT_VFDOutputs."ToMCAx[2]Deceleration" := UINT_TO_INT(#iUDT_VFDConfiguration.SpeedAxis.Deceleration * 10);

	            // Manual mode enable
	            IF #iqUDT_ConveyorInterface.ManualModeActive
	            THEN
	                #qUDT_VFDOutputs.ToMCActiveOpMode := #ci_ManualMode;
	            END_IF;

	            // Servo ON
	            IF #iUDT_VFDInputs.FromMCActiveOpMode = #ci_ManualMode
	                AND #iUDT_VFDInputs."FromMCAx[2]".Ready
	            THEN
	                #qUDT_VFDOutputs."ToMCAx[2]".Servo_ON := TRUE;
	            END_IF;

	            // Servo active
	            IF #iUDT_VFDInputs."FromMCAx[2]".Servo_active
	            THEN

	                IF #iUDT_VFDInputs.FromMCActiveOpMode = #ci_ManualMode
	                THEN
	                    // In manual mode jog outpus are used
	                    #qUDT_VFDOutputs."ToMCAx[2]".Jog_Fwd := NOT #sx_SpeedChange AND #iUDT_VFDConfiguration.SpeedAxis.InterlockFwd AND #iqUDT_ConveyorInterface.RunFwd;
	                    #qUDT_VFDOutputs."ToMCAx[2]".Jog_Bkwd := NOT #sx_SpeedChange AND #iUDT_VFDConfiguration.SpeedAxis.InterlockRvs AND #iqUDT_ConveyorInterface.RunRvs;
	                ELSE
	                    // In auto mode system command are used
	                    #qUDT_VFDOutputs.ToMCControl2.Ax_BeltRunFwd := #iUDT_VFDConfiguration.SpeedAxis.InterlockFwd AND #iqUDT_ConveyorInterface.RunFwd;
	                    #qUDT_VFDOutputs.ToMCControl2.Ax_BeltRunBkwd := #iUDT_VFDConfiguration.SpeedAxis.InterlockRvs AND #iqUDT_ConveyorInterface.RunRvs;
	                END_IF;
	            END_IF;
	        END_IF;

	        // Speed change reset
	        #sx_SpeedChange := FALSE;

	    END_REGION

	    REGION 7.4 - Bypasss mode

	        #qUDT_VFDOutputs.ToMCControl1.Bypass := #iqUDT_PolisorterInterface.BypassMode;

	    END_REGION

	END_REGION

	REGION 8 - Maintenance Mode

	    #iqUDT_PolisorterInterface.MaintenanceMode := #sx_HardwareAvailable
	    AND #iUDT_VFDInputs.FromMCActiveOpMode >= 10;

	    #sUDT_HMIStatus.MaintenanceWarning := #iqUDT_PolisorterInterface.MaintenanceMode;

	    #sUDT_HMIStatus.MaintenanceManualActiveWarning := #sx_HardwareAvailable
	    AND #iUDT_VFDInputs.FromMCActiveOpMode = #ci_MaintenanceManualMode;

	    #sUDT_HMIStatus.HomingActiveWarning := #sx_HardwareAvailable
	    AND #iUDT_VFDInputs.FromMCActiveOpMode = #ci_MaintenanceHoming;

	    #sUDT_HMIStatus.StressTestActiveWarning := #sx_HardwareAvailable
	    AND #iUDT_VFDInputs.FromMCActiveOpMode = #ci_MaintenanceStressTest;

	END_REGION

	REGION 9 - Statistics

	    // Profinet slave not online errors statistics

	    #sR_TRIG_PNSlaveNotOnline(CLK := #sUDT_HMIStatus.PNSlaveNotOnline);

	    IF #iqUDT_PolisorterInterface.ResetStatistics OR
	        #sUDT_HMIStatus.PNSlaveNotOnline
	    THEN

	        "FC_Statistics"(ix_Reset := #iqUDT_PolisorterInterface.ResetStatistics,
	                        ix_Activate := #sUDT_HMIStatus.PNSlaveNotOnline,
	                        ix_RTrigActivate := #sR_TRIG_PNSlaveNotOnline.Q,
	                        iqUDT_Statistics := #iqUDT_VFDStatistics.PNSlaveNotOnline);
	    END_IF;

	    // Profinet slave errors statistics

	    #sR_TRIG_PNSlaveError(CLK := #sUDT_HMIStatus.PNSlaveError);
	    IF #iqUDT_PolisorterInterface.ResetStatistics OR
	        #sUDT_HMIStatus.PNSlaveError
	    THEN

	        "FC_Statistics"(ix_Reset := #iqUDT_PolisorterInterface.ResetStatistics,
	                        ix_Activate := #sUDT_HMIStatus.PNSlaveError,
	                        ix_RTrigActivate := #sR_TRIG_PNSlaveError.Q,
	                        iqUDT_Statistics := #iqUDT_VFDStatistics.PNSlaveError);

	    END_IF;

	    // Axis 1 internal error statistics

	    #sR_TRIG_Ax1_InternalError(CLK := #sUDT_HMIStatus.Axis1InternalError);

	    IF #iqUDT_PolisorterInterface.ResetStatistics OR
	        #sUDT_HMIStatus.Axis1InternalError
	    THEN

	        "FC_Statistics"(ix_Reset := #iqUDT_PolisorterInterface.ResetStatistics,
	                        ix_Activate := #sUDT_HMIStatus.Axis1InternalError,
	                        ix_RTrigActivate := #sR_TRIG_Ax1_InternalError.Q,
	                        iqUDT_Statistics := #iqUDT_VFDStatistics.Ax1InternalError);

	    END_IF;

	    // Axis 2 internal error statistics

	    #sR_TRIG_Ax2_InternalError(CLK := #sUDT_HMIStatus.Axis2InternalError);

	    IF #iqUDT_PolisorterInterface.ResetStatistics OR
	        #sUDT_HMIStatus.Axis2InternalError
	    THEN

	        "FC_Statistics"(ix_Reset := #iqUDT_PolisorterInterface.ResetStatistics,
	                        ix_Activate := #sUDT_HMIStatus.Axis2InternalError,
	                        ix_RTrigActivate := #sR_TRIG_Ax2_InternalError.Q,
	                        iqUDT_Statistics := #iqUDT_VFDStatistics.Ax2InternalError);

	    END_IF;

	    // Communication error statistics

	    #sR_TRIG_CommunicationError(CLK := #sUDT_HMIStatus.CommunicationError);

	    IF #iqUDT_PolisorterInterface.ResetStatistics OR
	        #sUDT_HMIStatus.CommunicationError
	    THEN

	        "FC_Statistics"(ix_Reset := #iqUDT_PolisorterInterface.ResetStatistics,
	                        ix_Activate := #sUDT_HMIStatus.CommunicationError,
	                        ix_RTrigActivate := #sR_TRIG_CommunicationError.Q,
	                        iqUDT_Statistics := #iqUDT_VFDStatistics.CommunicationError);

	    END_IF;

	    // Axis 1 running statistics

	    #sR_TRIG_Ax1_Running(CLK := #iUDT_VFDInputs.FromMCStatus1.Running);

	    IF #iqUDT_PolisorterInterface.ResetStatistics OR
	        #iUDT_VFDInputs.FromMCStatus1.Running
	    THEN

	        "FC_Statistics"(ix_Reset := #iqUDT_PolisorterInterface.ResetStatistics,
	                        ix_Activate := #iUDT_VFDInputs.FromMCStatus1.Running,
	                        ix_RTrigActivate := #sR_TRIG_Ax1_Running.Q,
	                        iqUDT_Statistics := #iqUDT_VFDStatistics.Ax1Running);

	    END_IF;

	    // Axis 2 running statistics

	    #sR_TRIG_Ax2_Running(CLK := #iqUDT_ConveyorInterface.VFDRunning);

	    IF #iqUDT_PolisorterInterface.ResetStatistics OR
	        #iqUDT_ConveyorInterface.VFDRunning
	    THEN

	        "FC_Statistics"(ix_Reset := #iqUDT_PolisorterInterface.ResetStatistics,
	                        ix_Activate := #iqUDT_ConveyorInterface.VFDRunning,
	                        ix_RTrigActivate := #sR_TRIG_Ax2_Running.Q,
	                        iqUDT_Statistics := #iqUDT_VFDStatistics.Ax2Running);

	    END_IF;

	END_REGION

	REGION 10 - Status

	    #qUDT_HMIStatus := #sUDT_HMIStatus;

	END_REGION

	REGION 11 - Write interface outputs

	    // Axis 1 internal Error
	    #iqUDT_PolisorterInterface.InternalErrorVFD := #sx_Ax1_ErrorActive;

	    // Axis 1 internal Warning
	    #iqUDT_PolisorterInterface.InternalWarningVFD := #sx_Ax1_WarningActive;

	    // Axis 1 motor running
	    #iqUDT_PolisorterInterface.MotorRunning := #iUDT_VFDInputs.FromMCStatus1.Running;

	    // Axis 1 referenced
	    #iqUDT_PolisorterInterface.Referenced := #iUDT_VFDInputs.FromMCStatus1.Homed;

	    // Axis 1 positioning
	    #iqUDT_PolisorterInterface.Positioning := #iUDT_VFDInputs."FromMCAx[1]".Positioning
	    AND NOT #iUDT_VFDInputs."FromMCAx[1]".Standstill
	    AND NOT #iUDT_VFDInputs."FromMCAx[1]".Positioned;

	    // Axis 2 actual speed
	    #iqUDT_ConveyorInterface.ActualSpeed := REAL_TO_INT(#sr_Ax2ActualSpeed);

	    // Axis 2 internal Error
	    #iqUDT_ConveyorInterface.InternalErrorVFD := #iUDT_VFDInputs."FromMCAx[2]".Fault;

	    // Axis 2 motor running
	    #iqUDT_ConveyorInterface.VFDRunning := #sr_Ax2ActualSpeed > 0;

	    // Axis 2 at speed
	    #iqUDT_ConveyorInterface.VFDatSpeed := #sr_Ax2ActualSpeed < #iqUDT_ConveyorInterface.SpeedSetpoint + #iUDT_VFDConfiguration.SpeedAxis.SpeedSetpointWindow
	    AND #sr_Ax2ActualSpeed > #iqUDT_ConveyorInterface.SpeedSetpoint - #iUDT_VFDConfiguration.SpeedAxis.SpeedSetpointWindow;

	END_REGION
END_FUNCTION_BLOCK

FUNCTION_BLOCK "FB_FedExDecodeUDS"
TITLE = FB_Decode
{ S7_Optimized_Access := 'TRUE' }
AUTHOR : MHSE
FAMILY : UPS_SpecificCommunication
VERSION : 3.0
// ATTRIBUTES
// AUTO_NUMBER = True
// BLOCK_NUMBER = 238
// END_ATTRIBUTES
//Function block to decode UPS messages.
   VAR_INPUT
      iUDT_FacilitySystem { ExternalAccessible := 'False'; ExternalVisible := 'False'; ExternalWritable := 'False'} : "UDT_FedExFacility";   // UDS System configuration
      iUDT_FacilityPLC { ExternalAccessible := 'False'; ExternalVisible := 'False'; ExternalWritable := 'False'} : "UDT_FedExFacility";   // LLC System configuration
      is_LastHost { ExternalAccessible := 'False'; ExternalVisible := 'False'; ExternalWritable := 'False'} : String;   // Last connected UDS SystemID
   END_VAR

